	    // At setpoint
	    IF #Enabled = TRUE THEN
	        #sTag.bAtSetpoint := NOT(#sTag.bOutput);
	    ELSE
	        #sTag.bAtSetpoint := FALSE;
	    END_IF;
	
	    // Controller fault
	    #sTag.bFault := FALSE;
	
	END_IF;
	
	// Mode
	IF #sTag.bManualOverride = TRUE THEN
	    #sTag.nMode := 3;
	ELSIF #sTag.bEnable = TRUE THEN
	    #sTag.nMode := 1;
	ELSE
	    #sTag.nMode := 0;
	END_IF;
	
	// Local outputs
	#bOutput := #sTag.bOutput;
	#bAtSetpoint := #sTag.bAtSetpoint;
	
	
END_FUNCTION_BLOCK

FUNCTION_BLOCK "fbHysteresis2"   // FB64, LAD
TITLE = fbHysteresis2
{ S7_Optimized_Access := 'TRUE' }
AUTHOR : Heaten
VERSION : 0.1
// Hysteresis function with bool inputs
// stored: AutoNumber true, IsIECCheckEnabled false, IsRetainMemResEnabled false, MemoryReserve 0, SetENOAutomatically false, UDAEnableTagReadback false
   VAR_INPUT
      bEnable : Bool;
      bHigh : Bool;
      bLow : Bool;
      bAbove : Bool;
      bReset : Bool;
   END_VAR
   VAR_OUTPUT
      bOut : Bool;
   END_VAR
   VAR
      State : Bool;
   END_VAR
   VAR_TEMP
      bStartSignal : Bool;
      bStopSignal : Bool;
   END_VAR
BEGIN

REGION Network 1 (SCL): Polarity of the control
   // Above = 1: when process state is "high" eg cooling, emptying, depressurizing
   // Above = 0: when precess state is "low" eg heating, filling, pressurizing
   IF #bAbove = TRUE THEN
       // emptying, cooling, depressurizing etc
       #bStartSignal := #bHigh;
       #bStopSignal := NOT(#bLow);
   ELSE
       // filling, heating, pressurizing etc
       #bStartSignal := NOT(#bLow);
       #bStopSignal := #bHigh;
   END_IF;
END_REGION

REGION Network 2: Switch ouput
   // Initial state = OFF
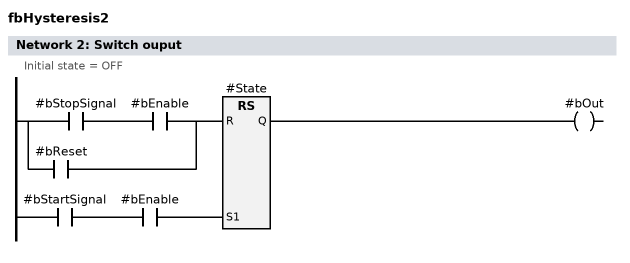
   RUNG wire#powerrail
      Contact( #bStopSignal )
      Contact( #bEnable )
      wire#w1
      S_RS(operand := #State, s1 := wire#w2)
      Coil( #bOut )
   END_RUNG
   RUNG wire#powerrail
      Contact( #bReset )
   END_RUNG wire#w1
   RUNG wire#powerrail
      Contact( #bStartSignal )
      Contact( #bEnable )
   END_RUNG wire#w2
   // the same network as SCL:
   IF (#bStopSignal AND #bEnable) OR #bReset THEN
       #State := FALSE;   // RS flip-flop
   END_IF;
   IF #bStartSignal AND #bEnable THEN #State := TRUE; END_IF;
   #bOut := #State;
END_REGION
END_FUNCTION_BLOCK

FUNCTION_BLOCK "ShaftSealCartridge"   // FB13, FBD
TITLE = Shaft seal cartridge
{ S7_Optimized_Access := 'TRUE' }
VERSION : 0.1
// stored: AutoNumber true, IsIECCheckEnabled false, IsRetainMemResEnabled false, MemoryReserve 100, SetENOAutomatically false, UDAEnableTagReadback false
   VAR_INPUT
      bEnable { ExternalAccessible := 'False'; ExternalVisible := 'False'; ExternalWritable := 'False'} : Bool;   // Enable from process. 1 = enabled, 0 = disabled.
      bReset { ExternalAccessible := 'False'; ExternalVisible := 'False'; ExternalWritable := 'False'} : Bool;
   END_VAR
   VAR
      Cooler { ExternalAccessible := 'False'; ExternalVisible := 'False'; ExternalWritable := 'False'} : "fbOnOffRegulator";
      Recharge { ExternalAccessible := 'False'; ExternalVisible := 'False'; ExternalWritable := 'False'; S7_SetPoint := 'True'} : "fbOnOffRegulator";
      A5257 { ExternalAccessible := 'False'; ExternalVisible := 'False'; ExternalWritable := 'False'; S7_SetPoint := 'True'} : "fbLowAlarm";
      A5258 { ExternalAccessible := 'False'; ExternalVisible := 'False'; ExternalWritable := 'False'; S7_SetPoint := 'True'} : "fbHighAlarm";
      A5259 { ExternalAccessible := 'False'; ExternalVisible := 'False'; ExternalWritable := 'False'; S7_SetPoint := 'True'} : "fbHighAlarm";
      A5260 { ExternalAccessible := 'False'; ExternalVisible := 'False'; ExternalWritable := 'False'; S7_SetPoint := 'True'} : "fbLowAlarm";
      A5261 { ExternalAccessible := 'False'; ExternalVisible := 'False'; ExternalWritable := 'False'; S7_SetPoint := 'True'} : "fbLowAlarm";
      A5262 { ExternalAccessible := 'False'; ExternalVisible := 'False'; ExternalWritable := 'False'; S7_SetPoint := 'True'} : "fbHighAlarm";
      A5263 { ExternalAccessible := 'False'; ExternalVisible := 'False'; ExternalWritable := 'False'; S7_SetPoint := 'True'} : "fbHighAlarm";
      A5268 { ExternalAccessible := 'False'; ExternalVisible := 'False'; ExternalWritable := 'False'; S7_SetPoint := 'True'} : "fbDigitalAlarm";
      nState { ExternalAccessible := 'False'; ExternalVisible := 'False'; ExternalWritable := 'False'; S7_SetPoint := 'True'} : USInt;
      bEnableAuto { ExternalAccessible := 'False'; ExternalVisible := 'False'; ExternalWritable := 'False'} : Bool;   // Circulation regulator is enabled in Auto
      bEnableCoolerAuto { ExternalAccessible := 'False'; ExternalVisible := 'False'; ExternalWritable := 'False'} : Bool;   // Cooling regulator is enabled in Auto
      bEnableRechargeAuto { ExternalAccessible := 'False'; ExternalVisible := 'False'; ExternalWritable := 'False'} : Bool;   // Recharging regulator is enabled in Auto
      bRunReqAuto { ExternalAccessible := 'False'; ExternalVisible := 'False'; ExternalWritable := 'False'} : Bool;   // Run in auto
      bStart { ExternalAccessible := 'False'; ExternalVisible := 'False'; ExternalWritable := 'False'} : R_TRIG;
   END_VAR
BEGIN

REGION Network 1: Delta-T over shaft seal
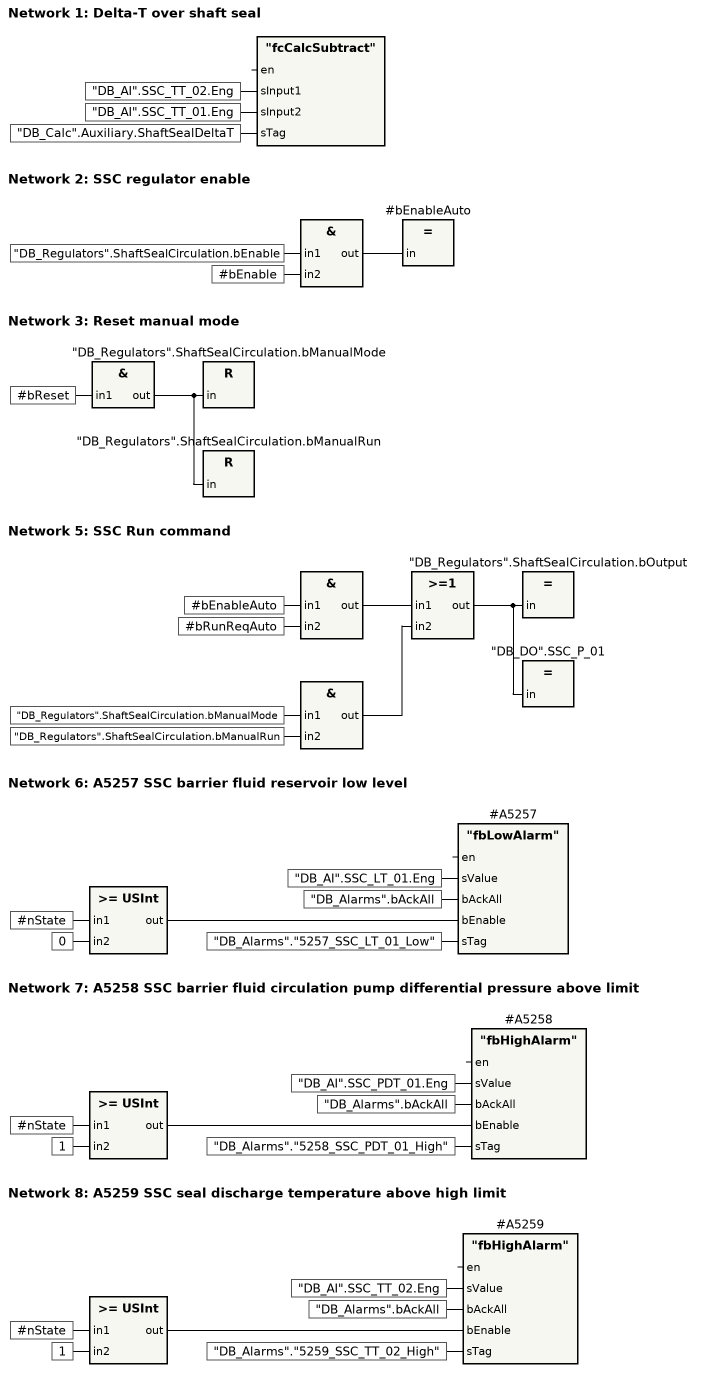
   "fcCalcSubtract"(sInput1 := "DB_AI".SSC_TT_02.Eng,
                    sInput2 := "DB_AI".SSC_TT_01.Eng,
                    sTag := "DB_Calc".Auxiliary.ShaftSealDeltaT);
END_REGION

REGION Network 2: SSC regulator enable
   // Start from input pin when enabled from HMI
   #bEnableAuto := "DB_Regulators".ShaftSealCirculation.bEnable AND #bEnable;
END_REGION

REGION Network 3: Reset manual mode
   IF #bReset THEN
       "DB_Regulators".ShaftSealCirculation.bManualMode := FALSE;
       "DB_Regulators".ShaftSealCirculation.bManualRun := FALSE;
   END_IF;
END_REGION

REGION Network 4 (SCL): SSC system state machine
   // Don't go into run state unless the pressure and temperature are first ok
   // Prevent retriggering
   #bStart(CLK := #bEnableAuto);

   CASE #nState OF

       0: // OFF
           #bEnableCoolerAuto := FALSE;
           #bEnableRechargeAuto := FALSE;
           #bRunReqAuto := FALSE;
           "DB_Regulators".ShaftSealCirculation.bFault := FALSE;
           IF #bStart.Q THEN
               #nState := 1;
           END_IF;
       1: // Startup. Wait for pressure and temperature to be ok
           #bEnableCoolerAuto := TRUE;
           #bEnableRechargeAuto := TRUE;
           //IF "DB_Regulators".ShaftSealCirculation.bEnable = FALSE THEN
           IF #bEnableAuto = FALSE THEN
               // Stop command
               #nState := 0;
           ELSIF "DB_Regulators".ShaftSealCirculation.bPressureLow AND "DB_Regulators".ShaftSealCirculation.bReservoirLow THEN
               // Barrier fluid pressure low and low fluid in recharge tank (can't recharge), give up.
               "DB_Regulators".ShaftSealCirculation.bFault := TRUE;
               #nState := 0;
           ELSIF "DB_Regulators".ShaftSealRecharge.bAtSetpoint AND "DB_Regulators".ShaftSealCooler.bAtSetpoint THEN
               // Pressure and temperature ok
               #nState := 2;
           END_IF;
       2: // Running
           #bRunReqAuto := TRUE;
           //IF "DB_Regulators".ShaftSealCirculation.bEnable = FALSE THEN
           IF #bEnableAuto = FALSE THEN
               // Stop command
               #nState := 0;
           END_IF;
           // Generate fault signal only in running state.
           "DB_Regulators".ShaftSealCirculation.bFault := "DB_Regulators".ShaftSealCirculation.bPressureLow OR "DB_Regulators".ShaftSealCirculation.bTemperatureHigh OR "DB_Regulators".ShaftSealCirculation.bDifferentialPressureHigh;
   END_CASE;
END_REGION

REGION Network 5: SSC Run command
   "DB_Regulators".ShaftSealCirculation.bOutput := (#bEnableAuto AND #bRunReqAuto) OR ("DB_Regulators".ShaftSealCirculation.bManualMode AND "DB_Regulators".ShaftSealCirculation.bManualRun);
   "DB_DO".SSC_P_01 := "DB_Regulators".ShaftSealCirculation.bOutput;
END_REGION

REGION Network 6: A5257 SSC barrier fluid reservoir low level
   // Always active
   #A5257(sValue := "DB_AI".SSC_LT_01.Eng,   // "fbLowAlarm"
          bAckAll := "DB_Alarms".bAckAll,
          bEnable := #nState >= 0,
          sTag := "DB_Alarms"."5257_SSC_LT_01_Low");
END_REGION

REGION Network 7: A5258 SSC barrier fluid circulation pump differential pressure above limit
   #A5258(sValue := "DB_AI".SSC_PDT_01.Eng,   // "fbHighAlarm"
          bAckAll := "DB_Alarms".bAckAll,
          bEnable := #nState >= 1,
          sTag := "DB_Alarms"."5258_SSC_PDT_01_High");
END_REGION

REGION Network 8: A5259 SSC seal discharge temperature above high limit
   #A5259(sValue := "DB_AI".SSC_TT_02.Eng,   // "fbHighAlarm"
          bAckAll := "DB_Alarms".bAckAll,
          bEnable := #nState >= 1,
          sTag := "DB_Alarms"."5259_SSC_TT_02_High");
END_REGION

REGION Network 9: A5260 SSC barrier fluid circulation pump suction temperature below low limit
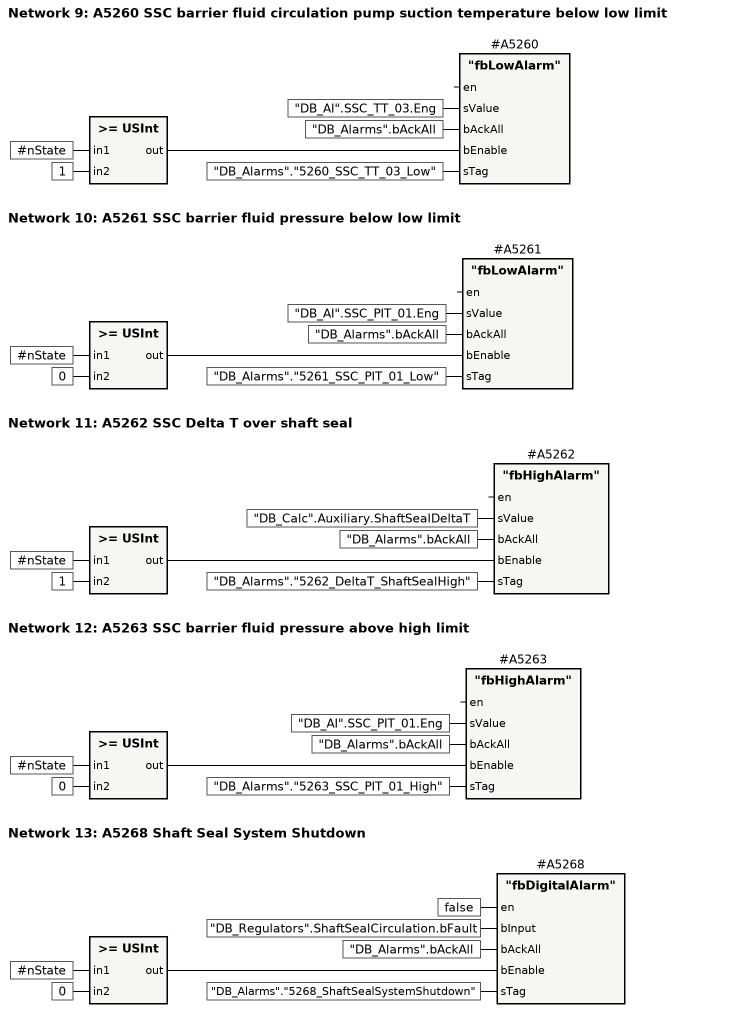
   #A5260(sValue := "DB_AI".SSC_TT_03.Eng,   // "fbLowAlarm"
          bAckAll := "DB_Alarms".bAckAll,
          bEnable := #nState >= 1,
          sTag := "DB_Alarms"."5260_SSC_TT_03_Low");
END_REGION

REGION Network 10: A5261 SSC barrier fluid pressure below low limit
   #A5261(sValue := "DB_AI".SSC_PIT_01.Eng,   // "fbLowAlarm"
          bAckAll := "DB_Alarms".bAckAll,
          bEnable := #nState >= 0,
          sTag := "DB_Alarms"."5261_SSC_PIT_01_Low");
END_REGION

REGION Network 11: A5262 SSC Delta T over shaft seal
   #A5262(sValue := "DB_Calc".Auxiliary.ShaftSealDeltaT,   // "fbHighAlarm"
          bAckAll := "DB_Alarms".bAckAll,
          bEnable := #nState >= 1,
          sTag := "DB_Alarms"."5262_DeltaT_ShaftSealHigh");
END_REGION

REGION Network 12: A5263 SSC barrier fluid pressure above high limit
   #A5263(sValue := "DB_AI".SSC_PIT_01.Eng,   // "fbHighAlarm"
          bAckAll := "DB_Alarms".bAckAll,
          bEnable := #nState >= 0,
          sTag := "DB_Alarms"."5263_SSC_PIT_01_High");
END_REGION

REGION Network 13: A5268 Shaft Seal System Shutdown
   // Regulator fault
   IF false THEN
       #A5268(bInput := "DB_Regulators".ShaftSealCirculation.bFault,   // "fbDigitalAlarm"
              bAckAll := "DB_Alarms".bAckAll,
              bEnable := #nState >= 0,
              sTag := "DB_Alarms"."5268_ShaftSealSystemShutdown");
   END_IF;
END_REGION

REGION Network 14: Faults
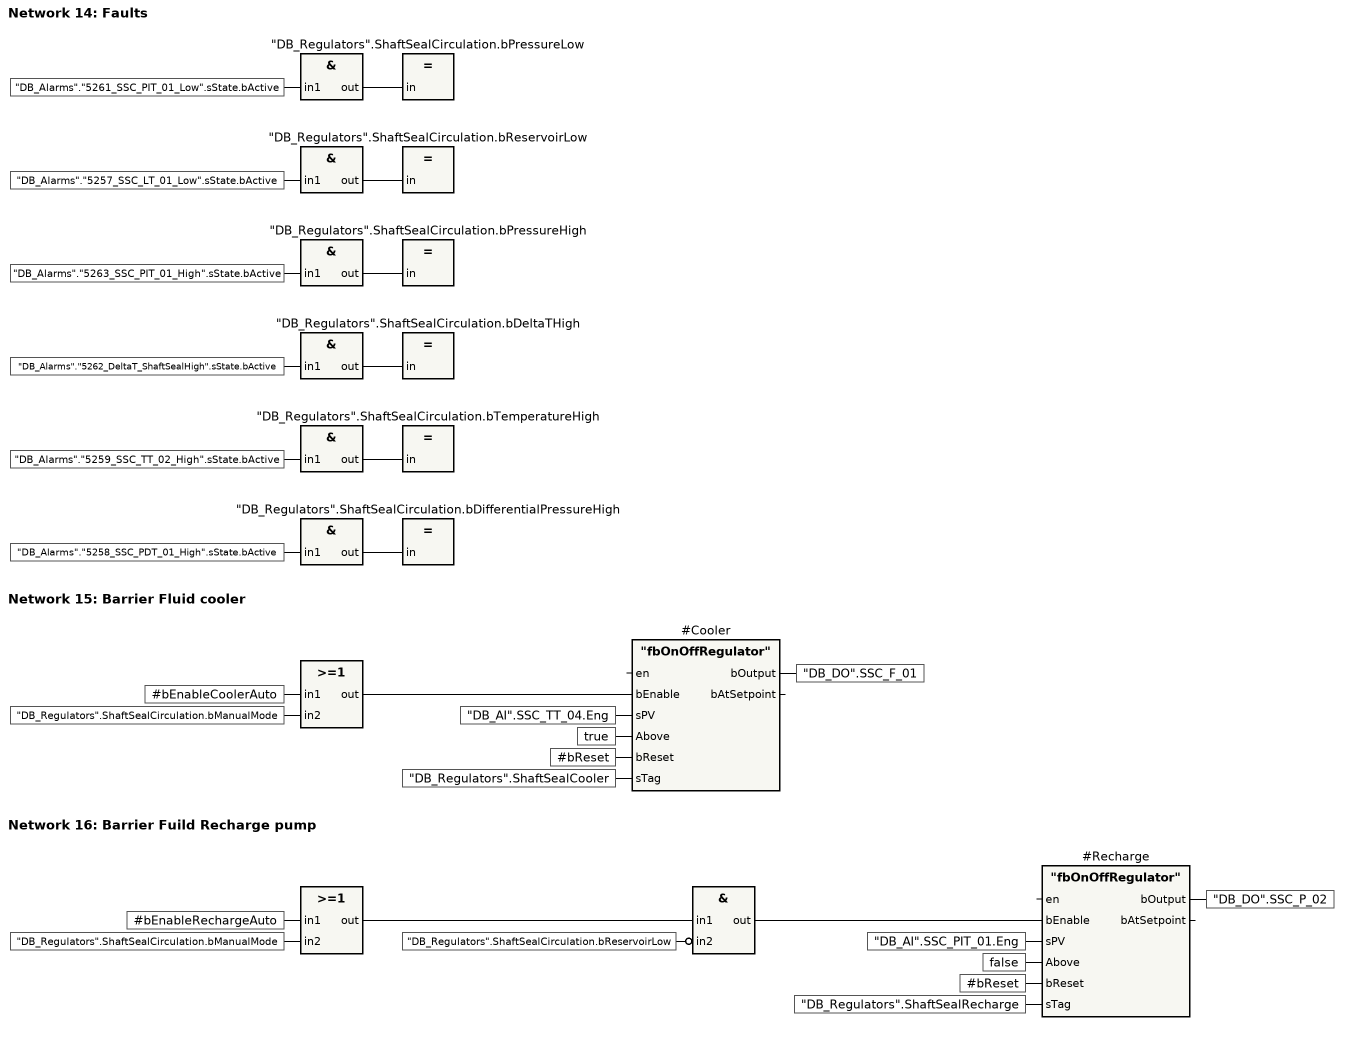
   "DB_Regulators".ShaftSealCirculation.bPressureLow := "DB_Alarms"."5261_SSC_PIT_01_Low".sState.bActive;
   "DB_Regulators".ShaftSealCirculation.bReservoirLow := "DB_Alarms"."5257_SSC_LT_01_Low".sState.bActive;
   "DB_Regulators".ShaftSealCirculation.bPressureHigh := "DB_Alarms"."5263_SSC_PIT_01_High".sState.bActive;
   "DB_Regulators".ShaftSealCirculation.bDeltaTHigh := "DB_Alarms"."5262_DeltaT_ShaftSealHigh".sState.bActive;
   "DB_Regulators".ShaftSealCirculation.bTemperatureHigh := "DB_Alarms"."5259_SSC_TT_02_High".sState.bActive;
   "DB_Regulators".ShaftSealCirculation.bDifferentialPressureHigh := "DB_Alarms"."5258_SSC_PDT_01_High".sState.bActive;
END_REGION

REGION Network 15: Barrier Fluid cooler
   // Run when the temperature in the barrier fluid gets too high
   #Cooler(bEnable := #bEnableCoolerAuto OR "DB_Regulators".ShaftSealCirculation.bManualMode,   // "fbOnOffRegulator"
           sPV := "DB_AI".SSC_TT_04.Eng,
           Above := true,
           bReset := #bReset,
           sTag := "DB_Regulators".ShaftSealCooler,
           bOutput => "DB_DO".SSC_F_01);
END_REGION

REGION Network 16: Barrier Fuild Recharge pump
   // Run when the pressure in the barrier fluid accumulator drops too low (and the reservoir is not empty)
   #Recharge(bEnable := (#bEnableRechargeAuto OR "DB_Regulators".ShaftSealCirculation.bManualMode) AND NOT "DB_Regulators".ShaftSealCirculation.bReservoirLow,   // "fbOnOffRegulator"
             sPV := "DB_AI".SSC_PIT_01.Eng,
             Above := false,
             bReset := #bReset,
             sTag := "DB_Regulators".ShaftSealRecharge,
             bOutput => "DB_DO".SSC_P_02);
END_REGION

REGION Network 17 (SCL)
   // Mode
   IF "DB_Regulators".ShaftSealCirculation.bManualMode = TRUE THEN
       "DB_Regulators".ShaftSealCirculation.nMode := 2;
   ELSIF "DB_Regulators".ShaftSealCirculation.bEnable = TRUE THEN
       "DB_Regulators".ShaftSealCirculation.nMode := 1;
   ELSE
       "DB_Regulators".ShaftSealCirculation.nMode := 0;
   END_IF;
END_REGION
END_FUNCTION_BLOCK

FUNCTION_BLOCK "LubricationPriming"   // FB20, FBD
{ S7_Optimized_Access := 'TRUE' }
VERSION : 0.1
// stored: AutoNumber true, IsIECCheckEnabled false, IsRetainMemResEnabled false, MemoryReserve 100, SetENOAutomatically false, UDAEnableTagReadback false
   VAR_INPUT
      bEnable { ExternalAccessible := 'False'; ExternalVisible := 'False'; ExternalWritable := 'False'} : Bool;
      bReset { ExternalAccessible := 'False'; ExternalVisible := 'False'; ExternalWritable := 'False'} : Bool;
   END_VAR
   VAR
      Pump { ExternalAccessible := 'False'; ExternalVisible := 'False'; ExternalWritable := 'False'} : "fbOnOffRegulator";
      Special { S7_SetPoint := 'True'} : "fbSpecialRegulator";
   END_VAR
   VAR_TEMP
      bOutput : Bool;
   END_VAR
BEGIN

REGION Network 1: Pump regulator
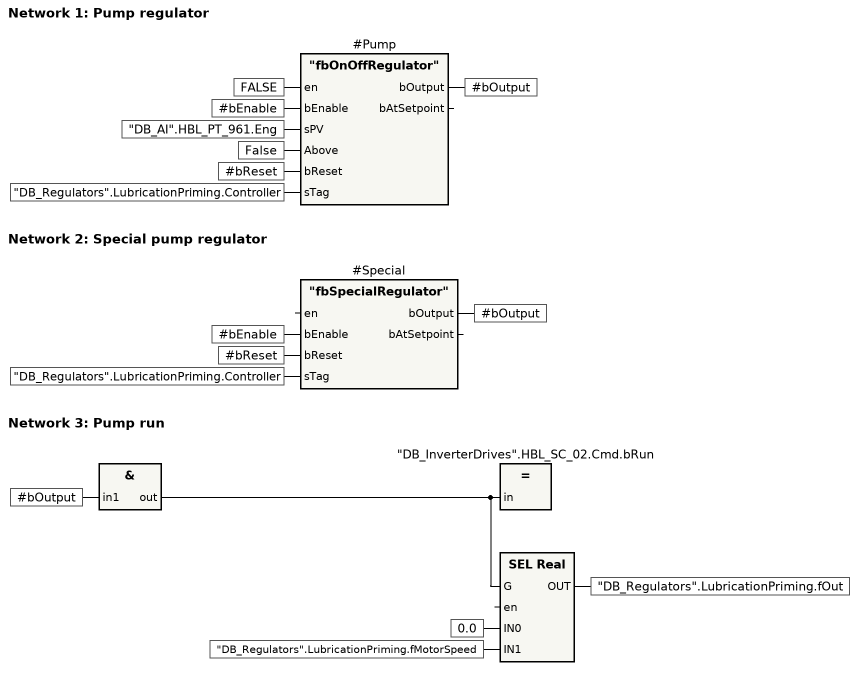
   IF FALSE THEN
       #Pump(bEnable := #bEnable,   // "fbOnOffRegulator"
             sPV := "DB_AI".HBL_PT_961.Eng,
             Above := False,
             bReset := #bReset,
             sTag := "DB_Regulators".LubricationPriming.Controller,
             bOutput => #bOutput);
   END_IF;
END_REGION

REGION Network 2: Special pump regulator
   // ##TEST: special situations require special regulators!
   #Special(bEnable := #bEnable,   // "fbSpecialRegulator"
            bReset := #bReset,
            sTag := "DB_Regulators".LubricationPriming.Controller,
            bOutput => #bOutput);
END_REGION

REGION Network 3: Pump run
   "DB_InverterDrives".HBL_SC_02.Cmd.bRun := #bOutput;
   "DB_Regulators".LubricationPriming.fOut := SEL(G := #bOutput, IN0 := 0.0, IN1 := "DB_Regulators".LubricationPriming.fMotorSpeed);
END_REGION

REGION Network 4: Inverter run
END_REGION
END_FUNCTION_BLOCK

FUNCTION_BLOCK "fbSpecialRegulator"
{ S7_Optimized_Access := 'TRUE' }
VERSION : 0.1
   VAR_INPUT 
      bEnable : Bool;   // Enable from process. 1 = enabled, 0 = disabled
      bReset : Bool;   // 1 = reset manual modes
   END_VAR

   VAR_OUTPUT 
      bOutput : Bool;
      bAtSetpoint : Bool;
   END_VAR

   VAR_IN_OUT 
      sTag : "stOnOffRegulator";
   END_VAR

   VAR 
      Dummy : Bool;
   END_VAR

   VAR_TEMP 
      fSetpoint : Real;
      Enabled : Bool;
   END_VAR


BEGIN
	// Special regulator.
	// Looks like an on/off regulator but in "Auto" mode, runs as soon as it is enabled. A kind of "null" regulator
	// The reason for still using this block is to allow all the other functions of the regulator, like the manual
	// override functions, and Reset, to still work. Not optimized, just a hack.
	// 
	
	// Reset manual modes.
	IF #bReset THEN
	    #sTag.bManualMode := FALSE;
	    #sTag.fManualSetpoint := 0.0;
	    #sTag.bManualOverride := FALSE;
	    #sTag.bOverrideCmd := FALSE;
	END_IF;
	
	IF #sTag.bManualOverride = TRUE THEN
	    // In manual override, everything is awesome
	    #sTag.bAtSetpoint := TRUE;
	    #sTag.bFault := FALSE;
	    #sTag.bOutput := #sTag.bOverrideCmd;
	ELSE
	    // Enabled when enabled from process and from HMI (Auto), no manual mode
	    #Enabled := (#bEnable AND #sTag.bEnable);
	
	    // Run controller
	    IF #Enabled = TRUE THEN
	        #sTag.bOutput := TRUE;
	    ELSE
	        #sTag.bOutput  := FALSE;
	    END_IF;
	    
	    #sTag.bAtSetpoint := NOT (#sTag.bOutput);
	    
	    // Controller fault
	    #sTag.bFault := FALSE;
	
	END_IF;
	
	// Mode
	IF #sTag.bManualOverride = TRUE THEN
	    #sTag.nMode := 3;
	ELSIF #sTag.bManualMode = TRUE THEN
	    #sTag.nMode := 2;
	ELSIF #sTag.bEnable = TRUE THEN
	    #sTag.nMode := 1;
	ELSE
	    #sTag.nMode := 0;
	END_IF;
	
	// Local outputs
	#bOutput := #sTag.bOutput;
	#bAtSetpoint := #sTag.bAtSetpoint;
	
	
END_FUNCTION_BLOCK

FUNCTION_BLOCK "fbPurgeControl"
{ S7_Optimized_Access := 'TRUE' }
AUTHOR : Heaten
VERSION : 0.1
   VAR_INPUT 
      bEnable : Bool;   // 1 = enable, 0 = disable
      bRotationStopped : Bool;   // 1 = rotation stopped, 0 = rotating
      DeltaP : "stCalcValue";   // [kPa] 
      Speed : "stCalcValue";   // [rpm]
      fCycleTime : Real;
   END_VAR

   VAR_OUTPUT 
      bPurging : Bool;
      bSpinning : Bool;
      bDone : Bool := false;
   END_VAR

   VAR_IN_OUT 
      sTag : "stPurgeControl";
   END_VAR

   VAR 
      nState : Int;   // 0 = Idle, 1 = Purge, 2 = Ramp up, 3 = Spin, 4 = Ramp down, 5 = Reset
      PurgeTimer {InstructionName := 'TON_TIME'; LibVersion := '1.0'; S7_SetPoint := 'False'} : TON_TIME;   // How long to purge for
      SpinTimer {InstructionName := 'TON_TIME'; LibVersion := '1.0'} : TON_TIME;   // How long to spin for
      PumpStartTimer {InstructionName := 'TON_TIME'; LibVersion := '1.0'} : TON_TIME;   // How long to wait for the pump to start & generate pressure
      tRamp : Time;   // Time to ramp up to spin speed
      tSpin : Time;   // Time at full spin speed
      Start {InstructionName := 'R_TRIG'; LibVersion := '1.0'; S7_SetPoint := 'False'} : R_TRIG;
   END_VAR

   VAR_TEMP 
      bEnabled : Bool;
   END_VAR

   VAR CONSTANT 
      PrimingDelay : Time := T#4s;
   END_VAR


BEGIN
	// Purge controller
	// Run a compressor purge cycle:
	// 1. Repeat x times: (where x can be zero)
	//    a. Drain the suction manifold. Either for a certain amount of time, or look at the deltaP over the pump
	//    b. Spin the compressor to get the suction line to barf up a slug of liquid, with configurable ramp, speed and duration
	// 2. Drain the suction manifold. Either for a certain amount of time, or look at the deltaP over the pump
	// 3. bDone = TRUE
	// NOTE: "look at the deltaP over the pump" means run the pump for #PrimingDelay, then continue as long as pump delta P is not less than 
	// sTag.Purge.fPurgeDeltaP
	
	// Enable. Edge trigger to run it only once. bReset is like a momentary disable
	#bEnabled := #bEnable AND #sTag.bEnable AND NOT #sTag.bReset;
	#Start(CLK := #bEnable AND #sTag.bEnable);
	
	// Be quiet when not in operation
	IF #bEnabled = FALSE THEN
	    #sTag.bDone := FALSE;
	END_IF;
	
	// Run timers outside of the state machine so they run & reset properly
	#PurgeTimer(IN := (#nState = 1 OR #nState = 6), PT := #sTag.Purge.tPurgeTime);
	#SpinTimer(IN := (#nState = 3), PT := #tSpin);
	#PumpStartTimer(IN := ((#nState = 1 OR #nState = 6) AND #sTag.Purge.nPurgeType = 1), PT := #PrimingDelay);
	
	// Purge sequencer
	CASE #nState OF
	    0: // Idle
	        IF #Start.Q = TRUE THEN
	            IF #sTag.nPurgeCycles = 0 THEN
	                #nState := 6;
	            ELSE
	                #sTag.nPurgeCyclesRemaining := #sTag.nPurgeCycles;
	                #sTag.bDone := FALSE;
	                #tRamp := UDINT_TO_TIME(REAL_TO_UDINT((#sTag.Spin.fSpinSpeed/#sTag.Spin.fSpinRamp)*1000));
	                #tSpin := #sTag.Spin.tSpinTime - 2 * #tRamp;
	                #nState := 1;
	            END_IF;
	        END_IF;
	    1: // Purge
	        IF #bEnabled = FALSE THEN
	            #nState := 5;
	        ELSE
	            // Start purging
	            #sTag.bPurging := TRUE;
	            // Decide when to stop
	            IF #sTag.Purge.nPurgeType = 0 THEN
	                // Timer
	                IF #PurgeTimer.Q = TRUE THEN
	                    #sTag.bPurging := FALSE;
	                    #nState := 2;
	                END_IF;
	            ELSIF #sTag.Purge.nPurgeType = 1 THEN
	                // Delta P
	                IF #PumpStartTimer.Q AND (#DeltaP.fValue < #sTag.Purge.fPurgeDeltaP) THEN
	                    #sTag.bPurging := FALSE;
	                    #nState := 2;
	                END_IF;
	            END_IF;
	        END_IF;
	    2: // Ramp Up
	        "RampLimiter"(InputValue            := #sTag.Spin.fSpinSpeed,                                  
	                      "PositivChange per_s" := #sTag.Spin.fSpinRamp,
	                      "NegativChange per_s" := -#sTag.Spin.fSpinRamp,
	                      fCycleTime            := #fCycleTime,
	                      OutputValue           := #sTag.fSpinOut);
	        IF #bEnabled = FALSE THEN
	            #nState := 5;
	        ELSIF #Speed.fValue > #sTag.Spin.fSpinSpeed - 5 THEN
	            #nState := 3;
	        END_IF;
	    3: // Spin
	        IF #bEnabled = FALSE THEN
	            #nState := 5;
	        ELSIF #SpinTimer.Q = TRUE THEN
	            #nState := 4;
	        END_IF;
	    4: // Ramp down
	        "RampLimiter"(InputValue            := 0.0,                         
	                      "PositivChange per_s" := #sTag.Spin.fSpinRamp,
	                      "NegativChange per_s" := -#sTag.Spin.fSpinRamp,
	                      fCycleTime            := #fCycleTime,
	                      OutputValue           := #sTag.fSpinOut);
	        IF #bEnabled = FALSE THEN
	            #nState := 5;
	        ELSIF #bRotationStopped = TRUE THEN
	            #sTag.fSpinOut := 0;
	            #sTag.nPurgeCyclesRemaining := #sTag.nPurgeCyclesRemaining - 1;
	            IF #sTag.nPurgeCyclesRemaining = 0 THEN
	                #nState := 6;
	            ELSE
	                #nState := 1;
	            END_IF;
	        END_IF;
	    5: // Reset
	        #sTag.nPurgeCyclesRemaining := 0;
	        #sTag.bPurging := FALSE;
	        #sTag.fSpinOut := 0;
	        #sTag.bDone := TRUE;
	        #nState := 0;
	    6: // Last purge
	        IF #bEnabled = FALSE THEN
	            #nState := 5;
	        ELSE
	            // Start purging
	            #sTag.bPurging := TRUE;
	            // Decide when to stop
	            IF #sTag.Purge.nPurgeType = 0 THEN
	                // Timer
	                IF #PurgeTimer.Q = TRUE THEN
	                    #sTag.bPurging := FALSE;
	                    #nState := 5;
	                END_IF;
	            ELSIF #sTag.Purge.nPurgeType = 1 THEN
	                // Delta P
	                IF #PumpStartTimer.Q AND (#DeltaP.fValue < #sTag.Purge.fPurgeDeltaP) THEN
	                    #sTag.bPurging := FALSE;
	                    #nState := 5;
	                END_IF;
	            END_IF;
	        END_IF;
	END_CASE;
	
	// Mode
	IF #sTag.bEnable = TRUE THEN
	    #sTag.nMode := 1;
	ELSE
	    #sTag.nMode := 0;
	END_IF;
	
	// Local outputs     
	#bDone := #sTag.bDone;
	#bPurging := #sTag.bPurging;
	#bSpinning := #sTag.bSpinning := (#nState = 2 OR #nState = 3 OR #nState = 4);
END_FUNCTION_BLOCK

FUNCTION_BLOCK "fbFilterDryer"   // FB53, FBD
TITLE = Periodic regulator with a fixed setpoint output
{ S7_Optimized_Access := 'TRUE' }
AUTHOR : Heaten
VERSION : 0.1
// stored: AutoNumber true, IsIECCheckEnabled false, IsRetainMemResEnabled false, MemoryReserve 0, SetENOAutomatically false, UDAEnableTagReadback false
   VAR_INPUT
      bEnable : Bool;
      bReset : Bool;
   END_VAR
   VAR_OUTPUT
      bOut : Bool;
      fOut : Real;
   END_VAR
   VAR_IN_OUT
      sTag : "stFilterDryer";
   END_VAR
   VAR
      Controller : "fbPeriodicRegulator";
   END_VAR
   VAR_TEMP
      bOutput_1 : Bool;
   END_VAR
BEGIN

REGION Network 1: Run regulator
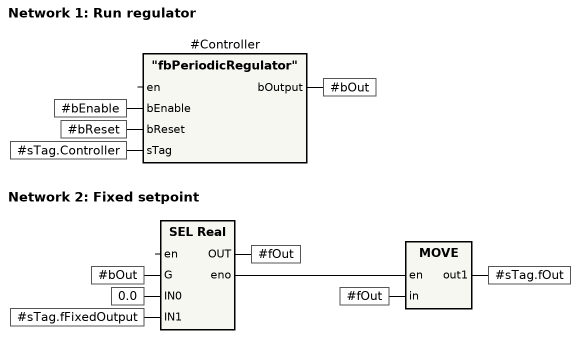
   #Controller(bEnable := #bEnable, bReset := #bReset, sTag := #sTag.Controller, bOutput => #bOut);   // "fbPeriodicRegulator"
END_REGION

REGION Network 2: Fixed setpoint
   // ENO of a box is taken as its EN; it also drops when the box reports an error
   #fOut := SEL(G := #bOut, IN0 := 0.0, IN1 := #sTag.fFixedOutput);
   #sTag.fOut := #fOut;
END_REGION
END_FUNCTION_BLOCK

FUNCTION_BLOCK "fbPeriodicRegulator"
{ S7_Optimized_Access := 'TRUE' }
AUTHOR : Heaten
VERSION : 0.1
   VAR_INPUT 
      bEnable : Bool;   // 1 = enable regulator, 0 = disable regulator
      bReset : Bool;   // 1 = reset everything to zero
   END_VAR

   VAR_OUTPUT 
      bOutput : Bool;
   END_VAR

   VAR_IN_OUT 
      sTag : "stPeriodicRegulator";
   END_VAR

   VAR 
      Controller { S7_SetPoint := 'False'} : "fbPWMController";
   END_VAR

   VAR_TEMP 
      Enabled : Bool;
   END_VAR


BEGIN
	// Periodic regulator
	// Periodic control of an output. Also called timer-based control.
	// The on-period and total period are parameters
	// Auto mode: periodic operation when Enable = true
	// Manual override: force the output on or off
	// 
	
	// Reset manual modes.
	IF #bReset THEN
	    #sTag.bManualOverride := FALSE;
	    #sTag.bOverrideCmd := FALSE;
	    #Controller.bEnable := FALSE;
	END_IF;
	
	// Select operating mode
	IF #sTag.bManualOverride = TRUE THEN
	    // In manual override, everything is awesome
	    #sTag.bFault := FALSE;
	    #sTag.bOutput := #sTag.bOverrideCmd;
	ELSE
	    // Enabled when enabled from process and from HMI (Auto)
	    #Enabled := (#bEnable AND #sTag.bEnable);
	    
	    // Run controller
	    #Controller(bEnable := #Enabled,
	                tOnTime := #sTag.tOnTime,
	                tPeriod := #sTag.tPeriod,
	                bOut => #sTag.bOutput,
	                tOnTimeElapsed => #sTag.tOnTimeElapsed,
	                tPeriodElapsed => #sTag.tPeriodElapsed);
	    
	    // Controller fault
	    #sTag.bFault := FALSE;
	    
	END_IF;
	
	// Mode
	IF #sTag.bManualOverride = TRUE THEN
	    #sTag.nMode := 3;
	ELSIF #sTag.bEnable = TRUE THEN
	    #sTag.nMode := 1;
	ELSE
	    #sTag.nMode := 0;
	END_IF;
	
	// Local outputs
	#bOutput := #sTag.bOutput;
END_FUNCTION_BLOCK

FUNCTION_BLOCK "fbOilRecovery"   // FB58, FBD
TITLE = Run once every X times with a fixed valve setpoint
{ S7_Optimized_Access := 'TRUE' }
AUTHOR : Heaten
VERSION : 0.1
// stored: AutoNumber true, IsIECCheckEnabled false, IsRetainMemResEnabled false, MemoryReserve 0, SetENOAutomatically false, UDAEnableTagReadback false
   VAR_INPUT
      bEnable : Bool;
      bReset : Bool;
   END_VAR
   VAR_OUTPUT
      bOut : Bool;
      fOut : Real;
   END_VAR
   VAR_IN_OUT
      sTag : "stOilRecovery";
   END_VAR
   VAR
      Controller : "fbOneShotRegulator";
      epEnabled : R_TRIG;
      RunCounter { S7_SetPoint := 'True'} : UInt;
      RunCounterMod : UInt;
   END_VAR
   VAR RETAIN
      Count { S7_SetPoint := 'True'} : Bool;
   END_VAR
   VAR_TEMP
      bEnabled : Bool;
   END_VAR
BEGIN

REGION Network 1: Run signal
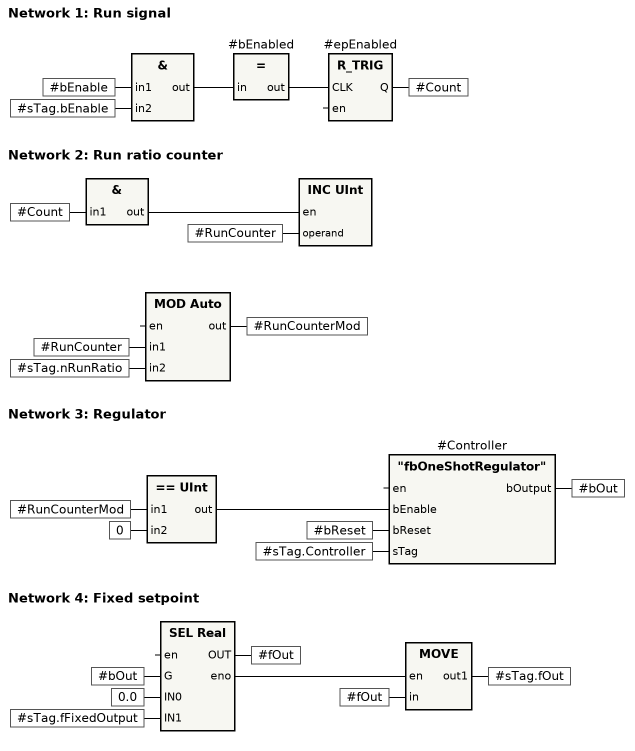
   #bEnabled := #bEnable AND #sTag.bEnable;
   #epEnabled(CLK := #bEnabled, Q => #Count);   // R_TRIG
END_REGION

REGION Network 2: Run ratio counter
   IF #Count THEN #RunCounter := #RunCounter + 1; END_IF;
   #RunCounterMod := #RunCounter MOD #sTag.nRunRatio;
END_REGION

REGION Network 3: Regulator
   // RunCounterMod is 0 every nth count.
   #Controller(bEnable := #RunCounterMod = 0, bReset := #bReset, sTag := #sTag.Controller, bOutput => #bOut);   // "fbOneShotRegulator"
END_REGION

REGION Network 4: Fixed setpoint
   // ENO of a box is taken as its EN; it also drops when the box reports an error
   #fOut := SEL(G := #bOut, IN0 := 0.0, IN1 := #sTag.fFixedOutput);
   #sTag.fOut := #fOut;
END_REGION
END_FUNCTION_BLOCK

FUNCTION_BLOCK "fbOneShotRegulator"
{ S7_Optimized_Access := 'TRUE' }
AUTHOR : Heaten
VERSION : 0.1
   VAR_INPUT 
      bEnable : Bool;   // 1 = enable regulator, 0 = disable regulator
      bReset : Bool;   // 1 = reset everything to zero
   END_VAR

   VAR_OUTPUT 
      bOutput : Bool;
   END_VAR

   VAR_IN_OUT 
      sTag : "stOneShotRegulator";
   END_VAR

   VAR 
      Controller { S7_SetPoint := 'False'} : "fbOneShot";
   END_VAR

   VAR_TEMP 
      Enabled : Bool;
   END_VAR


BEGIN
	// One-shot regulator
	// Activate something once for a certain period, with a start delay
	// The on-period and start delay are parameters
	// Auto mode: one-shot operation when Enable = true
	// Manual override: force the output on or off
	// 
	
	// Reset manual modes.
	IF #bReset THEN
	    #sTag.bManualOverride := FALSE;
	    #sTag.bOverrideCmd := FALSE;
	    #Controller.bEnable := FALSE;
	END_IF;
	
	// Select operating mode
	IF #sTag.bManualOverride = TRUE THEN
	    // In manual override, everything is awesome
	    #sTag.bFault := FALSE;
	    #sTag.bOutput := #sTag.bOverrideCmd;
	ELSE
	    // Enabled when enabled from process and from HMI (Auto)
	    #Enabled := (#bEnable AND #sTag.bEnable);
	    
	    // Run controller
	    #Controller(bEnable := #Enabled,
	                tOnTime := #sTag.tOnTime,
	                tStartDelay := #sTag.tStartDelay,
	                bOut => #sTag.bOutput,
	                tOnTimeElapsed => #sTag.tOnTimeElapsed,
	                tStartDelayElapsed => #sTag.tStartDelayElapsed);
	    
	    // Controller fault
	    #sTag.bFault := FALSE;
	    
	END_IF;
	
	// Mode
	IF #sTag.bManualOverride = TRUE THEN
	    #sTag.nMode := 3;
	ELSIF #sTag.bEnable = TRUE THEN
	    #sTag.nMode := 1;
	ELSE
	    #sTag.nMode := 0;
	END_IF;
	
	// Local outputs
	#bOutput := #sTag.bOutput;
END_FUNCTION_BLOCK

FUNCTION_BLOCK "fbOneShot"   // FB56, FBD
TITLE = One-shot with trigger delay
{ S7_Optimized_Access := 'TRUE' }
AUTHOR : Heaten
VERSION : 0.1
// stored: AutoNumber true, IsIECCheckEnabled false, IsRetainMemResEnabled false, MemoryReserve 0, SetENOAutomatically false, UDAEnableTagReadback false
   VAR_INPUT
      bEnable : Bool;   // 1 = enable controller, 0 = disable
      tOnTime : Time;
      tStartDelay : Time;
   END_VAR
   VAR_OUTPUT
      bOut : Bool;
      tOnTimeElapsed : Time;
      tStartDelayElapsed : Time;
   END_VAR
   VAR
      StartDelayTimer : TON_TIME;
      OnTimer { S7_SetPoint := 'True'} : TP_TIME;
   END_VAR
BEGIN

REGION Network 1: Trigger delay
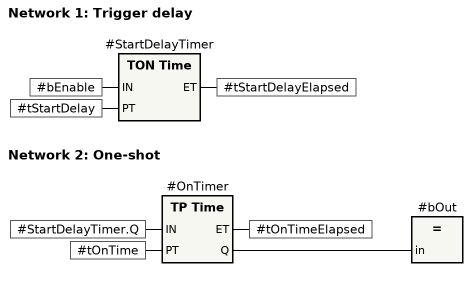
   #StartDelayTimer(IN := #bEnable, PT := #tStartDelay, ET => #tStartDelayElapsed);   // TON
END_REGION

REGION Network 2: One-shot
   #OnTimer(IN := #StartDelayTimer.Q, PT := #tOnTime, ET => #tOnTimeElapsed);   // TP
   #bOut := #OnTimer.Q;
END_REGION
END_FUNCTION_BLOCK

FUNCTION_BLOCK "fbNullRegulator"   // FB59, FBD
TITLE = PI Regulator
{ S7_Optimized_Access := 'TRUE' }
VERSION : 0.1
// stored: AutoNumber true, IsIECCheckEnabled false, IsRetainMemResEnabled false, MemoryReserve 0, SetENOAutomatically false, UDAEnableTagReadback false
   VAR_INPUT
      bEnable : Bool;
      bReset : Bool;
   END_VAR
   VAR_OUTPUT
      fOut : Real;
      bAtMin : Bool;
      bAtMax : Bool;
   END_VAR
   VAR_IN_OUT
      sTag : "stNullRegulator";
   END_VAR
   VAR
      Dummy : Real;
   END_VAR
   VAR_TEMP
      Enabled : Bool;
      fSelectedSetpoint : Real;
   END_VAR
BEGIN

REGION Network 1: Reset manual mode
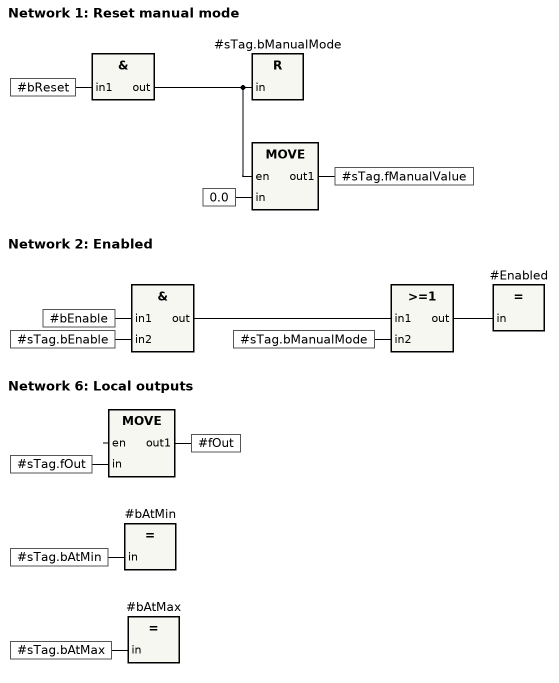
   IF #bReset THEN
       #sTag.bManualMode := FALSE;
       #sTag.fManualValue := 0.0;
   END_IF;
END_REGION

REGION Network 2: Enabled
   // Local input is from process control logic: when to run the regulator
   // Tag input is from HMI: do we want to run this regulator at all
   #Enabled := (#bEnable AND #sTag.bEnable) OR #sTag.bManualMode;
END_REGION

REGION Network 3 (SCL): Output selection
   IF #sTag.bManualMode = TRUE THEN
       #fSelectedSetpoint := #sTag.fManualValue;
   ELSE
       #fSelectedSetpoint := #sTag.fSetpoint;
   END_IF;

   #sTag.fOut := LIMIT(MN := #sTag.fOutMin, IN := #fSelectedSetpoint, MX := #sTag.fOutMax);
   #sTag.bAtMin := #sTag.fOut = #sTag.fOutMin;
   #sTag.bAtMax := #sTag.fOut = #sTag.fOutMax;
END_REGION

REGION Network 4 (SCL): Disable
   // This could be combined with logic above, and one day it might be!
   IF #Enabled = FALSE OR #sTag.bFault = TRUE THEN
       #sTag.fOut := 0.0;
       #sTag.bAtMin := FALSE;
       #sTag.bAtMax := FALSE;
   END_IF;
END_REGION

REGION Network 5 (SCL): Mode
   // Mode
   IF #sTag.bManualMode = TRUE THEN
       #sTag.nMode := 2;
   ELSIF #sTag.bEnable = TRUE THEN
       #sTag.nMode := 1;
   ELSE
       #sTag.nMode := 0;
   END_IF;
END_REGION

REGION Network 6: Local outputs
   #fOut := #sTag.fOut;
   #bAtMin := #sTag.bAtMin;
   #bAtMax := #sTag.bAtMax;
END_REGION
END_FUNCTION_BLOCK

FUNCTION_BLOCK "fbTrackingRegulator"
{ S7_Optimized_Access := 'TRUE' }
AUTHOR : Heaten
VERSION : 0.1
   VAR_INPUT 
      bEnable : Bool;
      bReset : Bool;
      sSP : "stCalcValue";   // Setpoint
      sPV : "stCalcValue";   // Process value
      sVelocity : "stCalcValue";   // Process value velocity
      fCycleTime : Real;
   END_VAR

   VAR_OUTPUT 
      fOut : Real;
      bAtMin : Bool;
      bAtMax : Bool;
   END_VAR

   VAR_IN_OUT 
      sTag : "stTrackingRegulator";
   END_VAR

   VAR 
      fStepsizePositive : Real;   // Output increment
      fStepsizeNegative : Real;   // Output decrement
   END_VAR

   VAR_TEMP 
      Enabled : Bool;
   END_VAR


BEGIN
	// Tracking regulator, a varaint of incremental control
	// Based on the "tracking ADC" algorithm, also known as "delta-encoded" or "counter-ramp"
	// The main parameters are the positive and negative slew rates. These control how big the increment in the output is.
	// The output is a staircase waveform which ramps the actuator up and down. The step size is calculated from the slew rate and cycle time.
	// There are two rates: the rate of change of the process value, and the rate of change of the actuator
	// For example, limiting the slew rate of a valve to keep the temperature increase below a limit
	
	// Detailed algorithm:
	// IF temperature < target AND temperature rate of change < positive limit THEN
	//    Increase valve output by positive step size
	// ELSIF temperature > target OR temperature rate of change > positive limit THEN
	//    Decrease valve output by negative step size
	// ELSE
	//    Keep valve output the same
	// END_IF
	// 
	
	// Tuning procedure:
	// 1. Set the fSlewRatePositive to something conservative like 0.2C/s
	// 2. Start HB and let it get to State 2
	// 3. Watch the heating of the steam condensers
	// 4. If the heating is very slow....
	
	// Copy to tag
	#sTag.fPV := #sPV.fValue;
	#sTag.fSP := #sSP.fValue;
	#sTag.fPVvelocity := #sVelocity.fValue;
	
	IF #bReset = TRUE THEN
	    #sTag.fOut := 0.0;
	    #sTag.bManualMode := FALSE;
	    #sTag.fManualValue := 0.0;
	END_IF;
	
	#Enabled := (#bEnable AND #sTag.bEnable) OR #sTag.bManualMode;
	
	// Step sizes
	#fStepsizePositive := #sTag.fSlewRatePositive / #fCycleTime;
	#fStepsizeNegative := #sTag.fSlewRateNegative / #fCycleTime;
	
	// Controller fault
	#sTag.bFault := #sSP.bError OR #sPV.bError OR #sVelocity.bError;
	
	IF #sTag.bManualMode = TRUE THEN
	    // Manual mode
	    #sTag.fOut := #sTag.fManualValue;
	ELSE
	    // Auto mode
	    IF #sPV.fValue < (#sSP.fValue - #sTag.fHysteresis) AND #sVelocity.fValue < #sTag.fVelocityPositiveLimit THEN
	        // Increase valve output
	        #sTag.fOut := #sTag.fOut + #fStepsizePositive;
	        #sTag.bAtSetpoint := FALSE;
	    ELSIF #sPV.fValue > (#sSP.fValue + #sTag.fHysteresis) OR #sVelocity.fValue > #sTag.fVelocityPositiveLimit THEN
	        // Decrease valve output
	        #sTag.fOut := #sTag.fOut - #fStepsizeNegative;
	        #sTag.bAtSetpoint := FALSE;
	    ELSE
	        // Keep valve output the same. Dummy branch but important to see the flow
	        #sTag.fOut := #sTag.fOut;
	        #sTag.bAtSetpoint := TRUE;
	    END_IF;
	END_IF;
	
	// Post processing
	IF #Enabled = FALSE OR #sTag.bFault = TRUE THEN
	    #sTag.fOut := 0.0;
	    #sTag.bAtMin := FALSE;
	    #sTag.bAtMax := FALSE;
	ELSE
	    //Evaluate limits exceeded first...
	    #sTag.bAtMin := NOT (#sTag.fOut > #sTag.fOutMin);
	    #sTag.bAtMax := #sTag.fOut >= #sTag.fOutMax;
	    //...before doing the actual limiting
	    #sTag.fOut := LIMIT(MN := #sTag.fOutMin, IN := #sTag.fOut, MX := #sTag.fOutMax);
	END_IF;
	
	// Mode
	IF #sTag.bManualMode = TRUE THEN
	    #sTag.nMode := 2;
	ELSIF #sTag.bEnable = TRUE THEN
	    #sTag.nMode := 1;
	ELSE
	    #sTag.nMode := 0;
	END_IF;
	
	// Local outputs
	#fOut := #sTag.fOut;
	#bAtMin := #sTag.bAtMin;
	#bAtMax := #sTag.bAtMax;
	
	
END_FUNCTION_BLOCK

FUNCTION_BLOCK "fbPIP_Regulator"   // FB28, FBD
TITLE = Position-velocity regulator (PI-P form)
{ S7_Optimized_Access := 'TRUE' }
AUTHOR : Heaten
VERSION : 0.1
// stored: AutoNumber true, IsIECCheckEnabled false, IsRetainMemResEnabled false, MemoryReserve 0, SetENOAutomatically false, UDAEnableTagReadback false
   VAR_INPUT
      sPV : "stCalcValue";   // Process value (position)
      sPVvel : "stCalcValue";   // Process value (velocity)
      fFeedback : Real;   // Output feedback (eg valve %, motor rpm)
      fCycleTime : Real;
      bEnable : Bool;
      bReset : Bool;
   END_VAR
   VAR_OUTPUT
      fOut : Real;
      bAtMin : Bool;
      bAtMax : Bool;
   END_VAR
   VAR_IN_OUT
      sTag : "stPIP_Regulator";
   END_VAR
   VAR
      Outer : Struct   // Outer loop = PI control
         D_Mem : Real;
         I_Mem : Real;
         Param_Mem : Real;
      END_STRUCT;
      Inner : Struct   // Inner loop = P control
         D_Mem : Real;
         I_Mem : Real;
         Param_Mem : Real;
      END_STRUCT;
      fSPVel : Real;
   END_VAR
   VAR_TEMP
      Enabled : Bool;
      fDeviation : Real;
      fDeviationVel : Real;
      bPI_AtMax : Bool;
      bPI_AtMin : Bool;
   END_VAR
BEGIN

REGION Network 1 (SCL): Comments and history
   // Position-velocity controller, cascaded PI-P form
   // 
   //                ___   pos   ____   vel   ___   vel   ___   out   __________         ______
   // pos ref ----> | Σ | ----> | PI | ----> | Σ | ----> | P | ----> | Actuator | ----> | Load |
   //             + |___| error |____|  ref  |___| error |___|       |__________|       |______|
   //                 ^ -                      ^ -                    _______               | 
   //                 |                        |_____________________| dP/dt |______________| measured velocity
   //                 |                                              |_______|              |
   //                 |_____________________________________________________________________| measured position
   //                 
   // For example, heating up a heat exchanger to a certain temperature without exceeding the temperature rise limit
   // 
   // Tuning Steps
   //
   // 1. Set the P constants of both controllers equal to 0, and integral to 9999. By default, the integral limit of the velocity
   //    controller should be set to the actuator's maximum position (eg 100%), and the integral limit of position
   //    controller should be set to the process max velocity (eg 5K/min).
   //
   // Important:from this step forth, the step response of position controller should always be evaluated.
   //
   // 2. Tune the KpVel parameter of the velocity controller. Increase the Kp of both position and velocity 
   //    controllers with a ratio of 10 (Kp_velocity = 10 * Kp_position). Once the real position starts to follow the
   //    reference position, stop increasing the Kp_position and only focus on increasing the Kp_velocity. Increase
   //    (sharpen) the velocity controller as much as possible. As a rule of thumb, increase kP_velocity until you get
   //    close to the instability margin (at this margin, you will feel a vibration effect and some acoustic noise
   //    which is because of controller sharpness). Now, you can reduce kP_velocity to 90% of its value to increase 
   //    the stability margin, and remove vibration noise.
   // 
   // 3. Now that the velocity controller is tuned, it is time to tune the parameters of the PID position 
   //    controller. Start with kP_position, and increase it until you again get close to the instability margin, and 
   //    then reduce kP_position to its 90%. So far, the proportional parts of both inner velocity loop and outer 
   //    position loop are tuned.
   //
   // 4. In this step, increase kI to eliminate the steady state error. As a suggestion start with kI equal to
   //    0.01, and in each step, increase it with a factor of 2. Increase kI step by step until the following two 
   //    conditions are met at the same time: - the overshoot is in its acceptable range - the steady-state error is 
   //    eliminated in a short enough period of time.
END_REGION

REGION Network 3: Reset manual mode
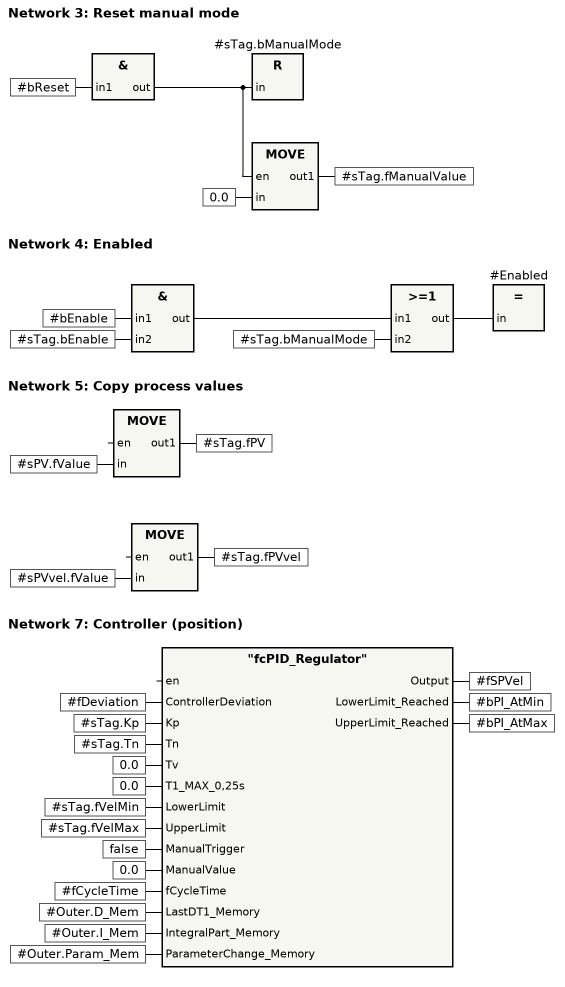
   IF #bReset THEN
       #sTag.bManualMode := FALSE;
       #sTag.fManualValue := 0.0;
   END_IF;
END_REGION

REGION Network 4: Enabled
   // Local input is from process control logic: when to run the regulator
   // Tag input is from HMI: do we want to run this regulator at all
   #Enabled := (#bEnable AND #sTag.bEnable) OR #sTag.bManualMode;
END_REGION

REGION Network 5: Copy process values
   #sTag.fPV := #sPV.fValue;
   #sTag.fPVvel := #sPVvel.fValue;
END_REGION

REGION Network 6 (SCL): Deviation (position)
   // NaN detection
   IF "isNaN"(#sTag.fSP) OR "isNaN"(#sTag.fPV) THEN
       #fDeviation := 0.0;
       #sTag.bFault := TRUE;
   ELSE
       #fDeviation := #sTag.fSP - #sTag.fPV;
       #sTag.bFault := FALSE;
   END_IF;
END_REGION

REGION Network 7: Controller (position)
   // NOTE: controller always runs regardless of mode.
   // This stage generates a velocity setpoint from the position error.
   // Max & min limits are of VELOCITY, this is not abug.
   "fcPID_Regulator"(ControllerDeviation := #fDeviation,
                     Kp := #sTag.Kp,
                     Tn := #sTag.Tn,
                     Tv := 0.0,
                     "T1_MAX_0,25s" := 0.0,
                     LowerLimit := #sTag.fVelMin,
                     UpperLimit := #sTag.fVelMax,
                     ManualTrigger := false,
                     ManualValue := 0.0,
                     fCycleTime := #fCycleTime,
                     LastDT1_Memory := #Outer.D_Mem,
                     IntegralPart_Memory := #Outer.I_Mem,
                     ParameterChange_Memory := #Outer.Param_Mem,
                     Output => #fSPVel,
                     LowerLimit_Reached => #bPI_AtMin,
                     UpperLimit_Reached => #bPI_AtMax);
END_REGION

REGION Network 8 (SCL): Deviation (velocity)
   // NaN detection
   IF "isNaN"(#sTag.fPVvel) THEN
       #fDeviationVel := 0.0;
       #sTag.bFault := TRUE;
   ELSE
       #fDeviationVel := #fSPVel - #sTag.fPVvel;
       #sTag.bFault := FALSE;
   END_IF;
END_REGION

REGION Network 9: Controller (velocity)
   // NOTE: controller always runs regardless of mode
   // This stage generates the manipulated value from the velocity error.
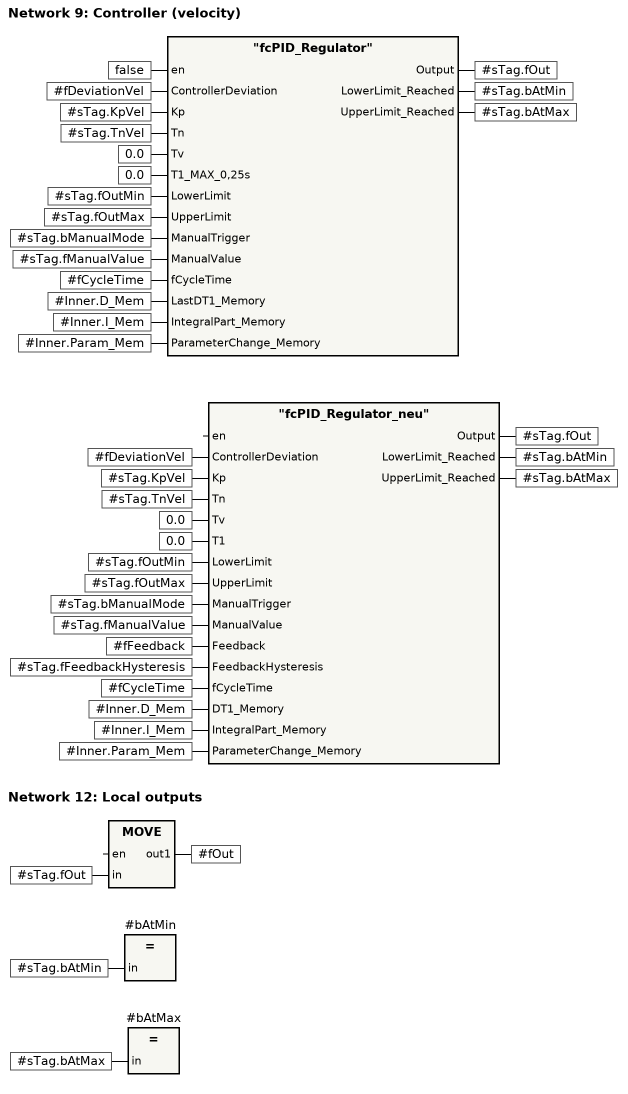
   IF false THEN
       "fcPID_Regulator"(ControllerDeviation := #fDeviationVel,
                         Kp := #sTag.KpVel,
                         Tn := #sTag.TnVel,
                         Tv := 0.0,
                         "T1_MAX_0,25s" := 0.0,
                         LowerLimit := #sTag.fOutMin,
                         UpperLimit := #sTag.fOutMax,
                         ManualTrigger := #sTag.bManualMode,
                         ManualValue := #sTag.fManualValue,
                         fCycleTime := #fCycleTime,
                         LastDT1_Memory := #Inner.D_Mem,
                         IntegralPart_Memory := #Inner.I_Mem,
                         ParameterChange_Memory := #Inner.Param_Mem,
                         Output => #sTag.fOut,
                         LowerLimit_Reached => #sTag.bAtMin,
                         UpperLimit_Reached => #sTag.bAtMax);
   END_IF;
   "fcPID_Regulator_neu"(ControllerDeviation := #fDeviationVel,
                         Kp := #sTag.KpVel,
                         Tn := #sTag.TnVel,
                         Tv := 0.0,
                         T1 := 0.0,
                         LowerLimit := #sTag.fOutMin,
                         UpperLimit := #sTag.fOutMax,
                         ManualTrigger := #sTag.bManualMode,
                         ManualValue := #sTag.fManualValue,
                         Feedback := #fFeedback,
                         FeedbackHysteresis := #sTag.fFeedbackHysteresis,
                         fCycleTime := #fCycleTime,
                         DT1_Memory := #Inner.D_Mem,
                         IntegralPart_Memory := #Inner.I_Mem,
                         ParameterChange_Memory := #Inner.Param_Mem,
                         Output => #sTag.fOut,
                         LowerLimit_Reached => #sTag.bAtMin,
                         UpperLimit_Reached => #sTag.bAtMax);
END_REGION

REGION Network 10 (SCL): Disable
   IF #Enabled = FALSE OR #sTag.bFault = TRUE THEN
       #sTag.fOut := 0.0;
       #sTag.bAtMin := FALSE;
       #sTag.bAtMax := FALSE;
   END_IF;
END_REGION

REGION Network 11 (SCL): Mode
   // Mode
   IF #sTag.bManualMode = TRUE THEN
       #sTag.nMode := 2;
   ELSIF #sTag.bEnable = TRUE THEN
       #sTag.nMode := 1;
   ELSE
       #sTag.nMode := 0;
   END_IF;
END_REGION

REGION Network 12: Local outputs
   #fOut := #sTag.fOut;
   #bAtMin := #sTag.bAtMin;
   #bAtMax := #sTag.bAtMax;
END_REGION
END_FUNCTION_BLOCK

FUNCTION_BLOCK "MotorControl"
{ S7_Optimized_Access := 'TRUE' }
VERSION : 0.1
   VAR_INPUT 
      PerformanceSetpoint { ExternalAccessible := 'False'; ExternalVisible := 'False'; ExternalWritable := 'False'} : Real;   // [%] Performance rate
      FastStop { ExternalAccessible := 'False'; ExternalVisible := 'False'; ExternalWritable := 'False'} : Bool;   // 1 = execute a fast stop, 0 = do nothing
   END_VAR

   VAR 
      NEngineRequest { ExternalAccessible := 'False'; ExternalVisible := 'False'; ExternalWritable := 'False'} : Real;   // [rpm]
      NEngineSetpoint { ExternalAccessible := 'False'; ExternalVisible := 'False'; ExternalWritable := 'False'} : Real;   // [rpm]
      InverterRun { ExternalAccessible := 'False'; ExternalVisible := 'False'; ExternalWritable := 'False'} : Bool;
      InverterReady { ExternalAccessible := 'False'; ExternalVisible := 'False'; ExternalWritable := 'False'} : Bool;
      HydrolockProtection { ExternalAccessible := 'False'; ExternalVisible := 'False'; ExternalWritable := 'False'} : Bool;
      A3400 { ExternalAccessible := 'False'; ExternalVisible := 'False'; ExternalWritable := 'False'; S7_SetPoint := 'False'} : "fbHMIEvent";
   END_VAR

   VAR_TEMP 
      PerformanceSetpointSelected : Real;   // [%] Selected performance setpoint
   END_VAR


BEGIN
	// Select motor setpoint and handle ready & run signals
	// NOTE: ramps are hardcoded, this is not ideal, should be in DB_CurrentSettings somewhere to make it easier to set up a new machine
	
	IF "DB_System".bEmergencyStop = TRUE THEN
	    #NEngineSetpoint := 0.0;
	ELSE
	    // Select setpoint
	    IF "DB_Regulators".PerformanceControl.ManualMode.ForcePowerSetpoint = TRUE THEN 
	        #PerformanceSetpointSelected := "DB_Regulators".PerformanceControl.ManualMode.ForcePowerSetpointValue;
	    ELSE
	        #PerformanceSetpointSelected := #"PerformanceSetpoint";
	    END_IF;
	
	    // Scale setpoint to RPM
	    #NEngineRequest := #PerformanceSetpointSelected / 100.0 * "DB_CurrentSetting".MissingSetting.Compressor.MaxOperationalSpeed;
	
	    // Limit setpoint
	    #NEngineRequest := LIMIT(IN := #NEngineRequest,
	                             MN := "DB_CurrentSetting".MissingSetting.Compressor.MinOperationalSpeed,
	                             MX := "DB_CurrentSetting".MissingSetting.Compressor.MaxOperationalSpeed);
	
	    CASE "DB_State".State.State_Number OF
	        0..1: // Init, offline modes
	            #NEngineSetpoint := 0.0;
	            #InverterReady := FALSE;
	            #InverterRun := FALSE;
	        2: // Standby
	            // If coming from one of the running modes, ramp down and stop
	            "RampLimiter"(InputValue            := 0.0,
	                          "PositivChange per_s" := 0.0,
	                          "NegativChange per_s" := -50.0,
	                          fCycleTime            := "DB_System".fCycleTime,
	                          OutputValue           := #NEngineSetpoint);
	            IF "DB_State".RunningConditions.CompressorStopped = TRUE THEN
	                #InverterReady := FALSE;
	                #InverterRun := FALSE;
	            END_IF;
	        3:  // PrepareStart
	            #NEngineSetpoint := 0.0;
	            #InverterReady := TRUE;
	        4:  // Start
	            IF "DB_State".RunningConditions.DoWarmStart = TRUE OR "DB_Regulators".PurgeControl.bDone = TRUE THEN
	                #InverterRun := TRUE;
	                // Preset the speed
	                #NEngineSetpoint := MAX(IN1 := #NEngineSetpoint, IN2 := "DB_CurrentSetting".MissingSetting.Compressor.MinStartupSpeed);   
	                "RampLimiter"(InputValue            := "DB_CurrentSetting".MissingSetting.System.HydrolockSpeed,                                  
	                              "PositivChange per_s" := 60.0,
	                              "NegativChange per_s" := -50.0,
	                              fCycleTime            := "DB_System".fCycleTime,
	                              OutputValue           := #NEngineSetpoint);
	            ELSE
	                // Note: Purge Control handles its own ramping
	                #NEngineSetpoint := "DB_Regulators".PurgeControl.fSpinOut;
	                #InverterRun := ("DB_Regulators".PurgeControl.nMode = 1);   // Don't touch
	            END_IF;
	
	            
	        5:  // Warmup
	            IF "DB_State".RunningConditions.RiskOfHydrolock = TRUE THEN
	                "RampLimiter"(InputValue            := MIN(IN1 := #NEngineSetpoint, IN2 := "DB_CurrentSetting".MissingSetting.System.HydrolockSpeed),
	                              "PositivChange per_s" := 0.0,
	                              "NegativChange per_s" := -500.0,
	                              fCycleTime            := "DB_System".fCycleTime,
	                              OutputValue           := #NEngineSetpoint);
	            ELSE
	                // Preset the speed
	                #NEngineSetpoint := MAX(IN1 := #NEngineSetpoint, IN2 := "DB_CurrentSetting".MissingSetting.Compressor.MinOperationalSpeed);
	                "RampLimiter"(InputValue := MIN(IN1 := "DB_CurrentSetting".MissingSetting.Compressor.WarmupSpeed, IN2 := #NEngineRequest),
	                              "PositivChange per_s" := 15.0,
	                              "NegativChange per_s" := -50.0,
	                              fCycleTime            := "DB_System".fCycleTime,
	                              OutputValue           := #NEngineSetpoint);
	            END_IF;
	        6:  // Running
	            IF "DB_State".RunningConditions.RiskOfHydrolock = TRUE THEN
	                "RampLimiter"(InputValue            := MIN(IN1 := #NEngineSetpoint, IN2 := "DB_CurrentSetting".MissingSetting.System.HydrolockSpeed),
	                              "PositivChange per_s" := 0.0,
	                              "NegativChange per_s" := -500.0,
	                              fCycleTime            := "DB_System".fCycleTime,
	                              OutputValue           := #NEngineSetpoint);
	            ELSE
	                "RampLimiter"(InputValue            := #NEngineRequest,
	                              "PositivChange per_s" := 30.0,
	                              "NegativChange per_s" := -30.0,
	                              fCycleTime            := "DB_System".fCycleTime,
	                              OutputValue           := #NEngineSetpoint);
	            END_IF;
	        7:  // Stopping
	            IF #FastStop = TRUE THEN
	                // Unconditional rampdown
	                "RampLimiter"(InputValue            := 0.0,
	                              "PositivChange per_s" := 0.0,
	                              "NegativChange per_s" := -500.0,
	                              fCycleTime            := "DB_System".fCycleTime,
	                              OutputValue           := #NEngineSetpoint);
	            ELSIF "DB_State".RunningConditions.SuctionLineDry = FALSE THEN
	                // Dry suction line at lower speed
	                "RampLimiter"(InputValue            := "DB_CurrentSetting".MissingSetting.Compressor.MinOperationalSpeed,
	                              "PositivChange per_s" := 60.0,
	                              "NegativChange per_s" := -50.0,
	                              fCycleTime            := "DB_System".fCycleTime,
	                              OutputValue           := #NEngineSetpoint);
	            ELSE
	                // Normal rampdown
	                "RampLimiter"(InputValue            := 0.0,
	                              "PositivChange per_s" := 0.0,
	                              "NegativChange per_s" := -50.0,
	                              fCycleTime            := "DB_System".fCycleTime,
	                              OutputValue           := #NEngineSetpoint);
	            END_IF;
	    END_CASE;
	
	END_IF;
	
	// Assign to inverter bits
	"DB_InverterDrives".HBL_SC_10.Cmd.bReady := #InverterReady;
	"DB_InverterDrives".HBL_SC_10.Cmd.bRun := #InverterRun;
	
END_FUNCTION_BLOCK

FUNCTION_BLOCK "ValveControl"   // FB27, FBD
TITLE = Setpoint selection & drivers
{ S7_Optimized_Access := 'TRUE' }
VERSION : 0.1
// stored: AutoNumber true, IsIECCheckEnabled false, IsRetainMemResEnabled false, MemoryReserve 100, SetENOAutomatically false, UDAEnableTagReadback false
   VAR_INPUT
      ValveSetpoint { ExternalAccessible := 'False'; ExternalVisible := 'False'; ExternalWritable := 'False'} : Real;   // [%] Valve position from regulator
   END_VAR
   VAR
      Setpoint { ExternalAccessible := 'False'; ExternalVisible := 'False'; ExternalWritable := 'False'} : Real;   // [%] Selected valve position
   END_VAR
   VAR_TEMP   // added for the SCL form of the ladder/FBD networks
      _w1 : Bool;
      _w2 : Bool;
   END_VAR
BEGIN

REGION Network 1 (SCL): Comment & history
   // Run valve drivers and do any switching of setpoints in case a valve is part of more than one control axis
END_REGION

REGION Network 2: Expansion valves
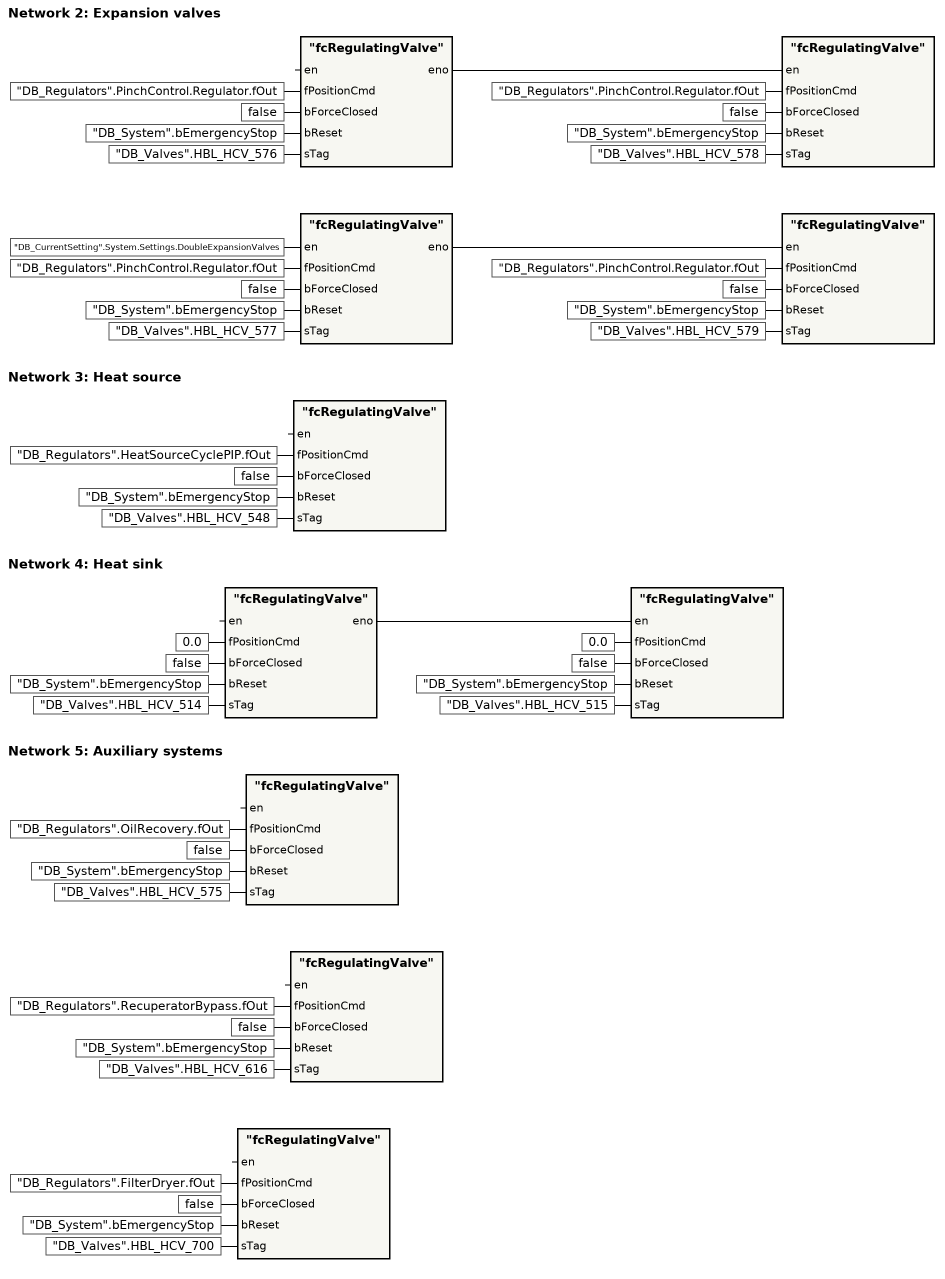
   "fcRegulatingValve"(fPositionCmd := "DB_Regulators".PinchControl.Regulator.fOut,
                       bForceClosed := false,
                       bReset := "DB_System".bEmergencyStop,
                       sTag := "DB_Valves".HBL_HCV_576,
                       ENO => #_w1);
   IF #_w1 THEN
       "fcRegulatingValve"(fPositionCmd := "DB_Regulators".PinchControl.Regulator.fOut,
                           bForceClosed := false,
                           bReset := "DB_System".bEmergencyStop,
                           sTag := "DB_Valves".HBL_HCV_578);
   END_IF;
   "fcRegulatingValve"(EN := "DB_CurrentSetting".System.Settings.DoubleExpansionValves,
                       fPositionCmd := "DB_Regulators".PinchControl.Regulator.fOut,
                       bForceClosed := false,
                       bReset := "DB_System".bEmergencyStop,
                       sTag := "DB_Valves".HBL_HCV_577,
                       ENO => #_w2);
   IF #_w2 THEN
       "fcRegulatingValve"(fPositionCmd := "DB_Regulators".PinchControl.Regulator.fOut,
                           bForceClosed := false,
                           bReset := "DB_System".bEmergencyStop,
                           sTag := "DB_Valves".HBL_HCV_579);
   END_IF;
END_REGION

REGION Network 3: Heat source
   "fcRegulatingValve"(fPositionCmd := "DB_Regulators".HeatSourceCyclePIP.fOut,
                       bForceClosed := false,
                       bReset := "DB_System".bEmergencyStop,
                       sTag := "DB_Valves".HBL_HCV_548);
END_REGION

REGION Network 4: Heat sink
   "fcRegulatingValve"(fPositionCmd := 0.0,
                       bForceClosed := false,
                       bReset := "DB_System".bEmergencyStop,
                       sTag := "DB_Valves".HBL_HCV_514,
                       ENO => #_w1);
   IF #_w1 THEN
       "fcRegulatingValve"(fPositionCmd := 0.0,
                           bForceClosed := false,
                           bReset := "DB_System".bEmergencyStop,
                           sTag := "DB_Valves".HBL_HCV_515);
   END_IF;
END_REGION

REGION Network 5: Auxiliary systems
   "fcRegulatingValve"(fPositionCmd := "DB_Regulators".OilRecovery.fOut,
                       bForceClosed := false,
                       bReset := "DB_System".bEmergencyStop,
                       sTag := "DB_Valves".HBL_HCV_575);
   "fcRegulatingValve"(fPositionCmd := "DB_Regulators".RecuperatorBypass.fOut,
                       bForceClosed := false,
                       bReset := "DB_System".bEmergencyStop,
                       sTag := "DB_Valves".HBL_HCV_616);
   "fcRegulatingValve"(fPositionCmd := "DB_Regulators".FilterDryer.fOut,
                       bForceClosed := false,
                       bReset := "DB_System".bEmergencyStop,
                       sTag := "DB_Valves".HBL_HCV_700);
END_REGION
END_FUNCTION_BLOCK

FUNCTION_BLOCK "fbSafetyRelay"
{ S7_Optimized_Access := 'TRUE' }
VERSION : 0.1
   VAR_INPUT 
      bStatus : Bool;   // Safety relay status 1 = ok, 0 = E-stop
   END_VAR

   VAR_OUTPUT 
      bExternalEstop : Bool;   // External E-stop is active
      bResetFailed : Bool;   // Failed to reset safety relay
   END_VAR

   VAR_IN_OUT 
      sTag : "stSafetyRelay";
   END_VAR

   VAR 
      SequenceTimer {InstructionName := 'TON_TIME'; LibVersion := '1.0'; S7_SetPoint := 'False'} : TON_TIME;
      ResetTimeout {InstructionName := 'TON_TIME'; LibVersion := '1.0'} : TON_TIME;
      ResetReq {InstructionName := 'R_TRIG'; LibVersion := '1.0'} : R_TRIG;   // Make sure command is an edge
   END_VAR


BEGIN
	// Sequencer to reset the safety relay.
	// 1. Close the PLC's E-stop loop output relay
	// 2. Send the reset command to the Safety relay
	// 3. Wait for a positive response, give up after timeout
	
	// Copy status into tag
	#sTag.bStatus := #bStatus;
	
	// Make reset signal an edge to prevent endless retriggering
	#ResetReq(CLK := #sTag.bResetReq);
	
	// Evaluate timers outside state machine so they reset properly
	#SequenceTimer(IN := (#sTag.nState = 1), PT := #sTag.tResetLoopTime);
	#ResetTimeout(IN := (#sTag.nState = 2), PT := #sTag.tResetTimeout);
	
	// Safety relay reset cycle
	CASE #sTag.nState OF
	    0: // Safety relay is tripped/open
	        IF #ResetReq.Q = TRUE THEN
	            #sTag.bResetLoop := TRUE;
	            #sTag.nState := 1;
	            #sTag.bResetFailed := FALSE;
	        ELSIF #bStatus = TRUE THEN
	            // Externally reset
	            #sTag.bResetFailed := FALSE;
	            #sTag.nState := 3;
	        END_IF;
	    1: // Give loop relay time to close
	        IF #SequenceTimer.Q = TRUE THEN 
	            #sTag.bResetCmd := TRUE;
	            #sTag.nState := 2;
	        END_IF;
	    2: // Wait for safety relay feedback or timeout
	        IF #bStatus = TRUE THEN
	            #sTag.bResetLoop := FALSE;
	            #sTag.bResetCmd := FALSE;
	            #sTag.nState := 3;
	        ELSIF #ResetTimeout.Q = TRUE THEN
	            #sTag.bResetLoop := FALSE;
	            #sTag.bResetCmd := FALSE;
	            #sTag.bResetFailed := TRUE;
	            #sTag.nState := 0;
	        END_IF;
	    3: // Safety relay is closed
	        IF #bStatus = FALSE THEN
	            #sTag.nState := 0;
	        END_IF;
	END_CASE;
	
	// Local outputs
	#bExternalEstop := NOT #bStatus;
	#bResetFailed := #sTag.bResetFailed;
	
END_FUNCTION_BLOCK

FUNCTION_BLOCK "StartStopControl"   // FB30, FBD
{ S7_Optimized_Access := 'TRUE' }
VERSION : 0.1
// stored: AutoNumber true, IsIECCheckEnabled false, IsRetainMemResEnabled false, MemoryReserve 0, SetENOAutomatically false, UDAEnableTagReadback false
   VAR_OUTPUT
      Run : Bool;   // 1 = run, 0 = stop
   END_VAR
   VAR
      StartRequestHMI { ExternalAccessible := 'False'; ExternalVisible := 'False'; ExternalWritable := 'False'; S7_SetPoint := 'True'} : R_TRIG;
      StartRequestApplication { ExternalAccessible := 'False'; ExternalVisible := 'False'; ExternalWritable := 'False'; S7_SetPoint := 'True'} : R_TRIG;
      StopRequestHMI { ExternalAccessible := 'False'; ExternalVisible := 'False'; ExternalWritable := 'False'; S7_SetPoint := 'True'} : R_TRIG;
      StopRequestApplication { ExternalAccessible := 'False'; ExternalVisible := 'False'; ExternalWritable := 'False'; S7_SetPoint := 'True'} : R_TRIG;
      EmergencyStopWaitTime { S7_SetPoint := 'True'} : TOF_TIME;
      StopRequestCriticalAlarm { S7_SetPoint := 'True'} : Bool;
   END_VAR
   VAR_TEMP
      StopRequestRegulatorFault : Bool;
   END_VAR
BEGIN

REGION Network 1: Start request signals
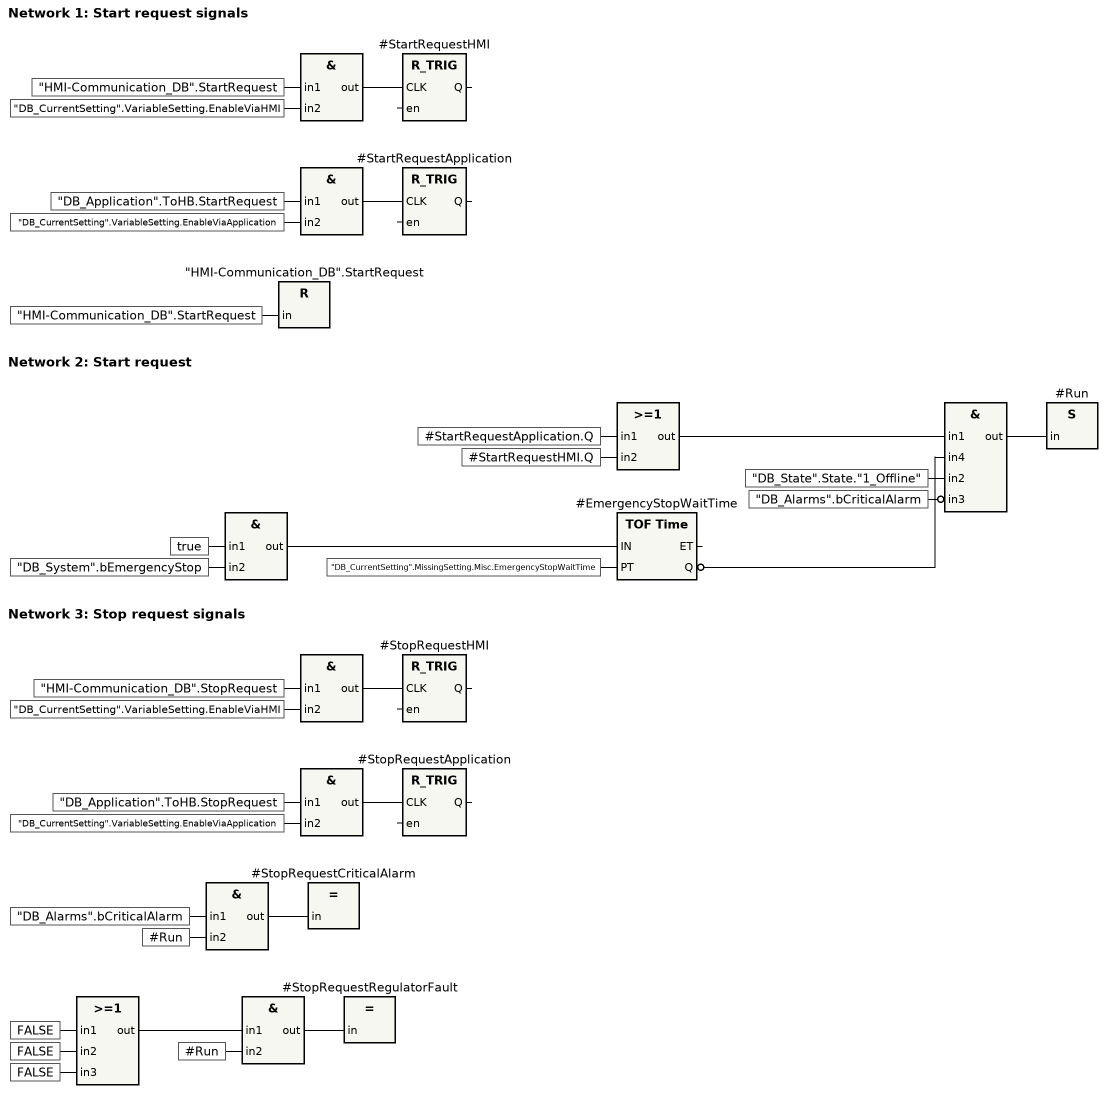
   #StartRequestHMI(CLK := "HMI-Communication_DB".StartRequest AND "DB_CurrentSetting".VariableSetting.EnableViaHMI);   // R_TRIG
   #StartRequestApplication(CLK := "DB_Application".ToHB.StartRequest AND "DB_CurrentSetting".VariableSetting.EnableViaApplication);   // R_TRIG
   IF "HMI-Communication_DB".StartRequest THEN "HMI-Communication_DB".StartRequest := FALSE; END_IF;
END_REGION

REGION Network 2: Start request
   // Start conditions:
   // 1. Start request from one of the control sources
   // 2. State 1 
   // 3. No critical alarms active
   // 4. E-stop lockout timer has expired
   // Also reset alarms
   #EmergencyStopWaitTime(IN := true AND "DB_System".bEmergencyStop,   // TOF
                          PT := "DB_CurrentSetting".MissingSetting.Misc.EmergencyStopWaitTime);
   IF (#StartRequestApplication.Q OR #StartRequestHMI.Q) AND NOT #EmergencyStopWaitTime.Q AND "DB_State".State."1_Offline" AND NOT "DB_Alarms".bCriticalAlarm THEN
       #Run := TRUE;
   END_IF;
END_REGION

REGION Network 3: Stop request signals
   // ##FIX decide what to do about regulator faults.
   #StopRequestHMI(CLK := "HMI-Communication_DB".StopRequest AND "DB_CurrentSetting".VariableSetting.EnableViaHMI);   // R_TRIG
   #StopRequestApplication(CLK := "DB_Application".ToHB.StopRequest AND "DB_CurrentSetting".VariableSetting.EnableViaApplication);   // R_TRIG
   #StopRequestCriticalAlarm := "DB_Alarms".bCriticalAlarm AND #Run;
   #StopRequestRegulatorFault := (FALSE OR FALSE OR FALSE) AND #Run;
END_REGION

REGION Network 4: Stop request
   // Stop condition is one of:
   // 1. Stop request from one of the control sources (HMI or App PLC)
   // 2. Forced into State 7 Stop (and the machine should follow)
   // 3. Critical Alarm
   // 4. Emergency Stop. (This is also technically a critical alarm but alarms can be disabled)
   // 5. Regulator fault
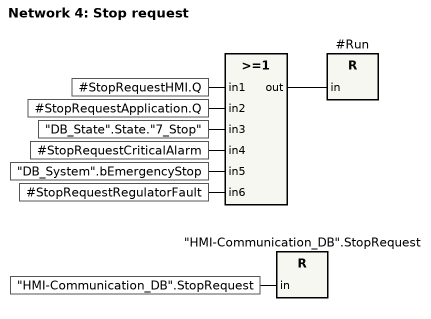
   IF #StopRequestHMI.Q OR #StopRequestApplication.Q OR "DB_State".State."7_Stop" OR #StopRequestCriticalAlarm OR "DB_System".bEmergencyStop OR #StopRequestRegulatorFault THEN
       #Run := FALSE;
   END_IF;
   IF "HMI-Communication_DB".StopRequest THEN "HMI-Communication_DB".StopRequest := FALSE; END_IF;
END_REGION
END_FUNCTION_BLOCK

FUNCTION_BLOCK "OutputProcessing"   // FB11, FBD
TITLE = Output mapping
{ S7_Optimized_Access := 'TRUE' }
VERSION : 0.1
// stored: AutoNumber true, IsIECCheckEnabled false, IsRetainMemResEnabled false, MemoryReserve 0, SetENOAutomatically false, UDAEnableTagReadback false
BEGIN

REGION Network 1: Digital
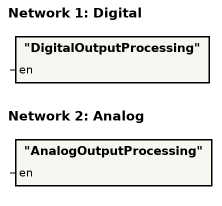
   "DigitalOutputProcessing"();
END_REGION

REGION Network 2: Analog
   "AnalogOutputProcessing"();
END_REGION
END_FUNCTION_BLOCK

FUNCTION "DigitalOutputProcessing" : Void   // FC11, FBD
TITLE = Output mapping
{ S7_Optimized_Access := 'TRUE' }
VERSION : 0.1
// stored: AutoNumber true, IsIECCheckEnabled false, SetENOAutomatically false, UDAEnableTagReadback false
   VAR_TEMP
      Spare : Bool;
   END_VAR
BEGIN

REGION Network 1: Emergency Stop output
   // 1 = ok, 0 = emergency stop
   // If emergency stop is not active, or you want to reset the safety relay, output is high.
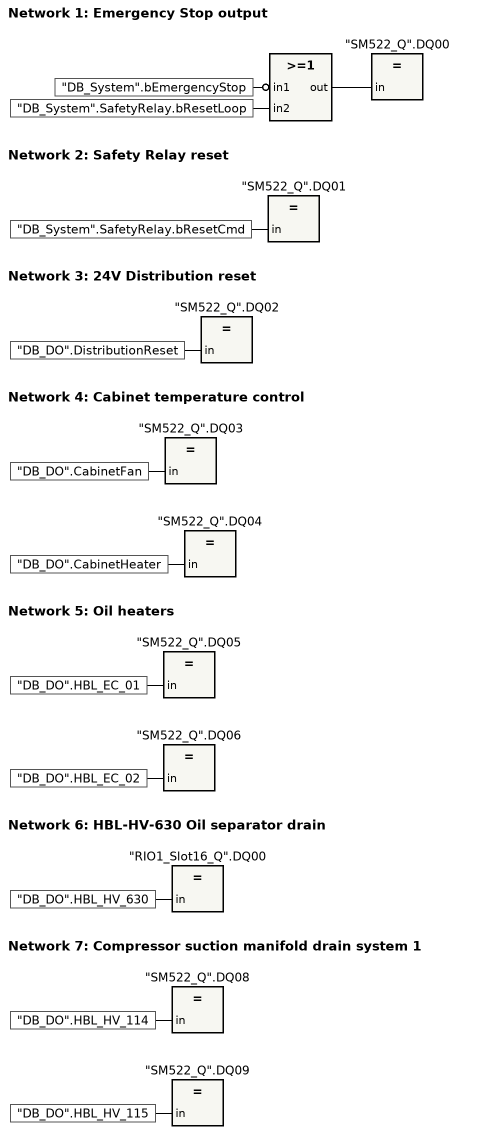
   "SM522_Q".DQ00 := NOT "DB_System".bEmergencyStop OR "DB_System".SafetyRelay.bResetLoop;
END_REGION

REGION Network 2: Safety Relay reset
   "SM522_Q".DQ01 := "DB_System".SafetyRelay.bResetCmd;
END_REGION

REGION Network 3: 24V Distribution reset
   "SM522_Q".DQ02 := "DB_DO".DistributionReset;
END_REGION

REGION Network 4: Cabinet temperature control
   "SM522_Q".DQ03 := "DB_DO".CabinetFan;
   "SM522_Q".DQ04 := "DB_DO".CabinetHeater;
END_REGION

REGION Network 5: Oil heaters
   "SM522_Q".DQ05 := "DB_DO".HBL_EC_01;
   "SM522_Q".DQ06 := "DB_DO".HBL_EC_02;
END_REGION

REGION Network 6: HBL-HV-630 Oil separator drain
   "RIO1_Slot16_Q".DQ00 := "DB_DO".HBL_HV_630;
END_REGION

REGION Network 7: Compressor suction manifold drain system 1
   // Valves directly from suction manifold to sump (optional)
   "SM522_Q".DQ08 := "DB_DO".HBL_HV_114;
   "SM522_Q".DQ09 := "DB_DO".HBL_HV_115;
END_REGION

REGION Network 8: Shaft Seal Cartridge (SSC)
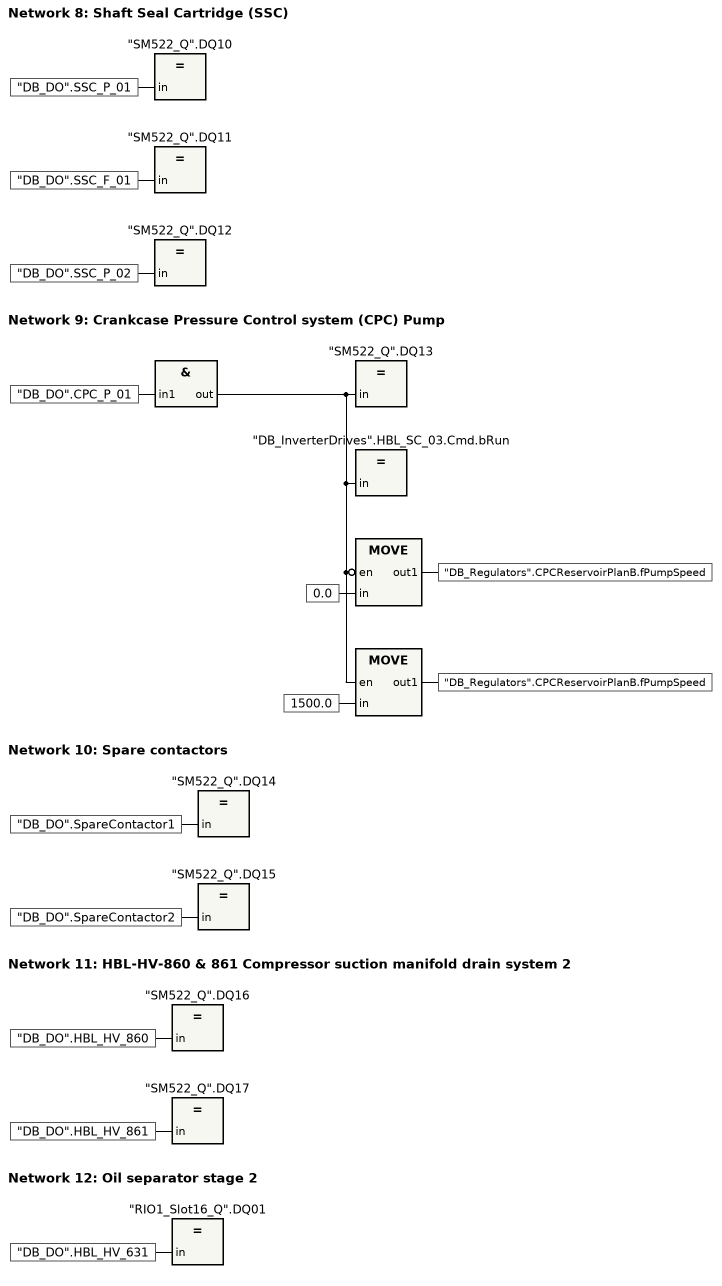
   "SM522_Q".DQ10 := "DB_DO".SSC_P_01;
   "SM522_Q".DQ11 := "DB_DO".SSC_F_01;
   "SM522_Q".DQ12 := "DB_DO".SSC_P_02;
END_REGION

REGION Network 9: Crankcase Pressure Control system (CPC) Pump
   // 10.02.2025 TSS: Normally DQ13, but now an inverter. And this is the ugly hack to make it work until we know how it really should be.
   "SM522_Q".DQ13 := "DB_DO".CPC_P_01;
   "DB_InverterDrives".HBL_SC_03.Cmd.bRun := "DB_DO".CPC_P_01;
   IF NOT "DB_DO".CPC_P_01 THEN "DB_Regulators".CPCReservoirPlanB.fPumpSpeed := 0.0; END_IF;
   IF "DB_DO".CPC_P_01 THEN "DB_Regulators".CPCReservoirPlanB.fPumpSpeed := 1500.0; END_IF;
END_REGION

REGION Network 10: Spare contactors
   "SM522_Q".DQ14 := "DB_DO".SpareContactor1;
   "SM522_Q".DQ15 := "DB_DO".SpareContactor2;
END_REGION

REGION Network 11: HBL-HV-860 & 861 Compressor suction manifold drain system 2
   // Valves to share the CPC system with the Purge controller
   "SM522_Q".DQ16 := "DB_DO".HBL_HV_860;
   "SM522_Q".DQ17 := "DB_DO".HBL_HV_861;
END_REGION

REGION Network 12: Oil separator stage 2
   "RIO1_Slot16_Q".DQ01 := "DB_DO".HBL_HV_631;
END_REGION

REGION Network 13: HBL-HV-640
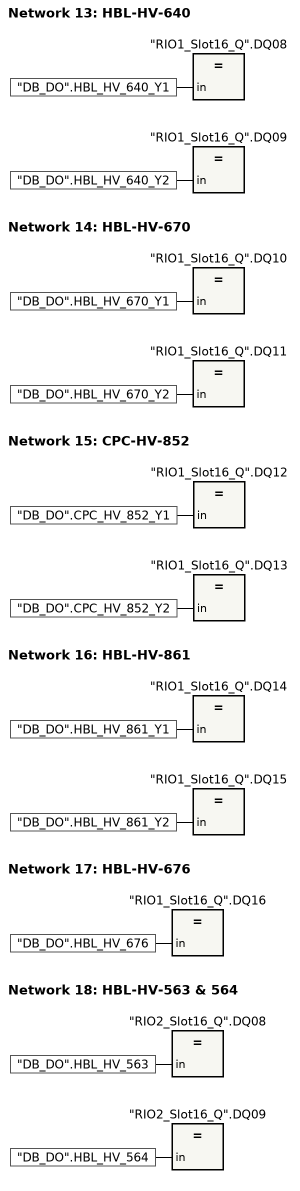
   "RIO1_Slot16_Q".DQ08 := "DB_DO".HBL_HV_640_Y1;
   "RIO1_Slot16_Q".DQ09 := "DB_DO".HBL_HV_640_Y2;
END_REGION

REGION Network 14: HBL-HV-670
   "RIO1_Slot16_Q".DQ10 := "DB_DO".HBL_HV_670_Y1;
   "RIO1_Slot16_Q".DQ11 := "DB_DO".HBL_HV_670_Y2;
END_REGION

REGION Network 15: CPC-HV-852
   "RIO1_Slot16_Q".DQ12 := "DB_DO".CPC_HV_852_Y1;
   "RIO1_Slot16_Q".DQ13 := "DB_DO".CPC_HV_852_Y2;
END_REGION

REGION Network 16: HBL-HV-861
   "RIO1_Slot16_Q".DQ14 := "DB_DO".HBL_HV_861_Y1;
   "RIO1_Slot16_Q".DQ15 := "DB_DO".HBL_HV_861_Y2;
END_REGION

REGION Network 17: HBL-HV-676
   "RIO1_Slot16_Q".DQ16 := "DB_DO".HBL_HV_676;
END_REGION

REGION Network 18: HBL-HV-563 & 564
   "RIO2_Slot16_Q".DQ08 := "DB_DO".HBL_HV_563;
   "RIO2_Slot16_Q".DQ09 := "DB_DO".HBL_HV_564;
END_REGION
END_FUNCTION

FUNCTION "AnalogOutputProcessing" : Void   // FC12, FBD
TITLE = Output mapping and scaling
{ S7_Optimized_Access := 'TRUE' }
VERSION : 0.1
// stored: AutoNumber true, IsIECCheckEnabled false, SetENOAutomatically false, UDAEnableTagReadback false
BEGIN

REGION Network 1: HBL-HCV-576
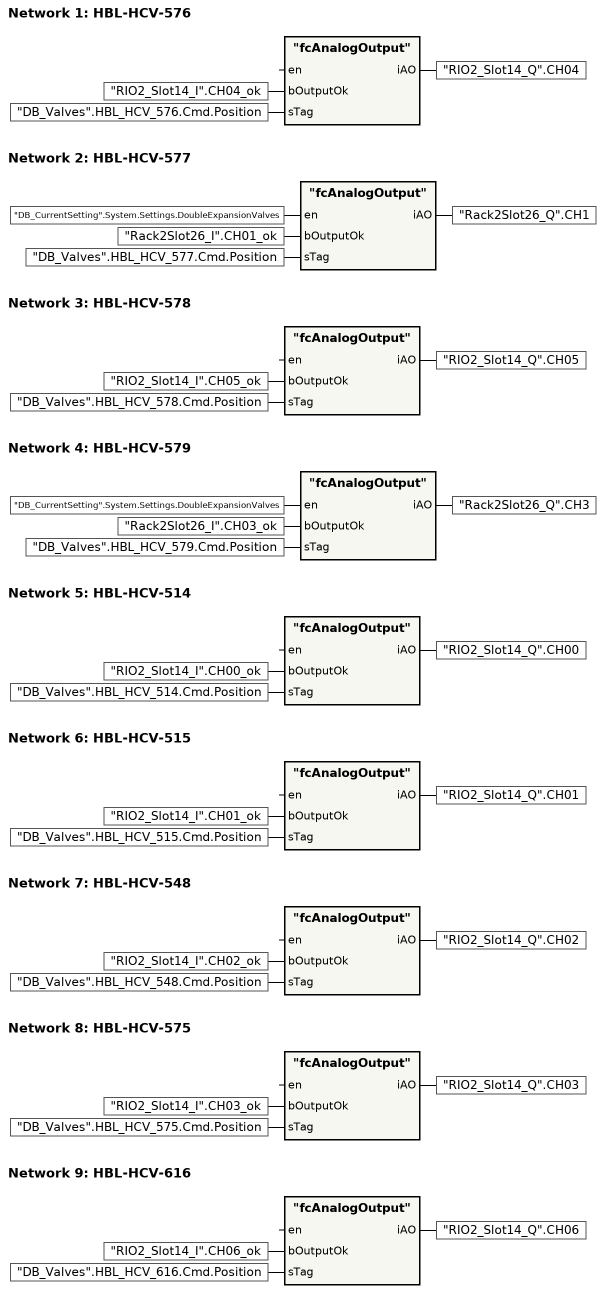
   "fcAnalogOutput"(bOutputOk := "RIO2_Slot14_I".CH04_ok,
                    sTag := "DB_Valves".HBL_HCV_576.Cmd.Position,
                    iAO => "RIO2_Slot14_Q".CH04);
END_REGION

REGION Network 2: HBL-HCV-577
   IF "DB_CurrentSetting".System.Settings.DoubleExpansionValves THEN
       "fcAnalogOutput"(bOutputOk := "Rack2Slot26_I".CH01_ok,
                        sTag := "DB_Valves".HBL_HCV_577.Cmd.Position,
                        iAO => "Rack2Slot26_Q".CH1);
   END_IF;
END_REGION

REGION Network 3: HBL-HCV-578
   "fcAnalogOutput"(bOutputOk := "RIO2_Slot14_I".CH05_ok,
                    sTag := "DB_Valves".HBL_HCV_578.Cmd.Position,
                    iAO => "RIO2_Slot14_Q".CH05);
END_REGION

REGION Network 4: HBL-HCV-579
   IF "DB_CurrentSetting".System.Settings.DoubleExpansionValves THEN
       "fcAnalogOutput"(bOutputOk := "Rack2Slot26_I".CH03_ok,
                        sTag := "DB_Valves".HBL_HCV_579.Cmd.Position,
                        iAO => "Rack2Slot26_Q".CH3);
   END_IF;
END_REGION

REGION Network 5: HBL-HCV-514
   "fcAnalogOutput"(bOutputOk := "RIO2_Slot14_I".CH00_ok,
                    sTag := "DB_Valves".HBL_HCV_514.Cmd.Position,
                    iAO => "RIO2_Slot14_Q".CH00);
END_REGION

REGION Network 6: HBL-HCV-515
   "fcAnalogOutput"(bOutputOk := "RIO2_Slot14_I".CH01_ok,
                    sTag := "DB_Valves".HBL_HCV_515.Cmd.Position,
                    iAO => "RIO2_Slot14_Q".CH01);
END_REGION

REGION Network 7: HBL-HCV-548
   "fcAnalogOutput"(bOutputOk := "RIO2_Slot14_I".CH02_ok,
                    sTag := "DB_Valves".HBL_HCV_548.Cmd.Position,
                    iAO => "RIO2_Slot14_Q".CH02);
END_REGION

REGION Network 8: HBL-HCV-575
   "fcAnalogOutput"(bOutputOk := "RIO2_Slot14_I".CH03_ok,
                    sTag := "DB_Valves".HBL_HCV_575.Cmd.Position,
                    iAO => "RIO2_Slot14_Q".CH03);
END_REGION

REGION Network 9: HBL-HCV-616
   "fcAnalogOutput"(bOutputOk := "RIO2_Slot14_I".CH06_ok,
                    sTag := "DB_Valves".HBL_HCV_616.Cmd.Position,
                    iAO => "RIO2_Slot14_Q".CH06);
END_REGION

REGION Network 10: HBL-HCV-700
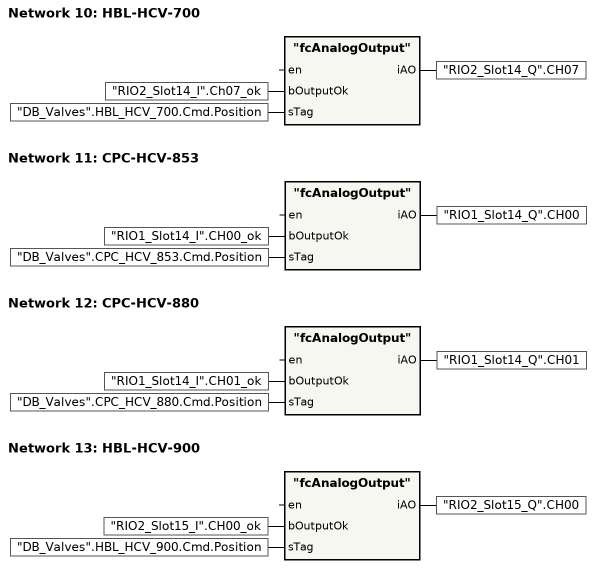
   "fcAnalogOutput"(bOutputOk := "RIO2_Slot14_I".Ch07_ok,
                    sTag := "DB_Valves".HBL_HCV_700.Cmd.Position,
                    iAO => "RIO2_Slot14_Q".CH07);
END_REGION

REGION Network 11: CPC-HCV-853
   "fcAnalogOutput"(bOutputOk := "RIO1_Slot14_I".CH00_ok,
                    sTag := "DB_Valves".CPC_HCV_853.Cmd.Position,
                    iAO => "RIO1_Slot14_Q".CH00);
END_REGION

REGION Network 12: CPC-HCV-880
   "fcAnalogOutput"(bOutputOk := "RIO1_Slot14_I".CH01_ok,
                    sTag := "DB_Valves".CPC_HCV_880.Cmd.Position,
                    iAO => "RIO1_Slot14_Q".CH01);
END_REGION

REGION Network 13: HBL-HCV-900
   "fcAnalogOutput"(bOutputOk := "RIO2_Slot15_I".CH00_ok,
                    sTag := "DB_Valves".HBL_HCV_900.Cmd.Position,
                    iAO => "RIO2_Slot15_Q".CH00);
END_REGION
END_FUNCTION

FUNCTION_BLOCK "Diagnosis"   // FB1, FBD
TITLE = Misc alarm handling
{ S7_Optimized_Access := 'TRUE' }
VERSION : 0.1
// stored: AutoNumber true, IsIECCheckEnabled false, IsRetainMemResEnabled false, MemoryReserve 0, SetENOAutomatically false, UDAEnableTagReadback false
   VAR
      A0001 { ExternalAccessible := 'False'; ExternalVisible := 'False'; ExternalWritable := 'False'} : "fbHMIEvent";
      A1002 { ExternalAccessible := 'False'; ExternalVisible := 'False'; ExternalWritable := 'False'; S7_SetPoint := 'True'} : "fbHMIEvent";
      A1003 { ExternalAccessible := 'False'; ExternalVisible := 'False'; ExternalWritable := 'False'; S7_SetPoint := 'True'} : "fbHMIEvent";
   END_VAR
BEGIN

REGION Network 1: 0001 Watchdog timeout OB1
   // "DB_Alarms"."0001_WatchdogTimeoutOB1".bInput is written by OB80, but alarm is processed here (OB80 is not cyclic)
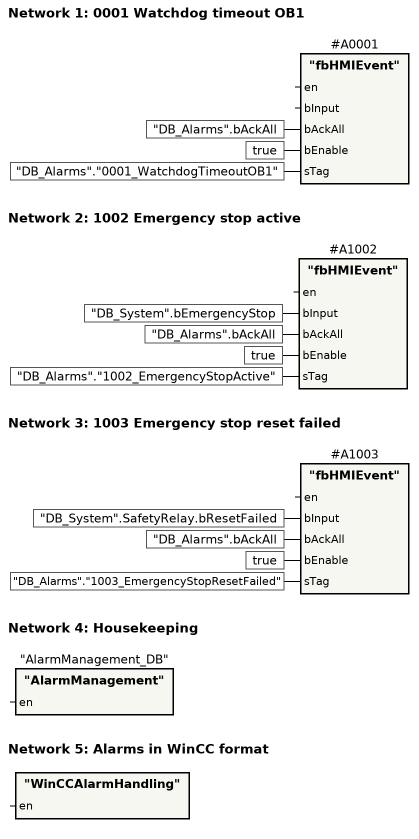
   #A0001(bAckAll := "DB_Alarms".bAckAll, bEnable := true, sTag := "DB_Alarms"."0001_WatchdogTimeoutOB1");   // "fbHMIEvent"
END_REGION

REGION Network 2: 1002 Emergency stop active
   #A1002(bInput := "DB_System".bEmergencyStop,   // "fbHMIEvent"
          bAckAll := "DB_Alarms".bAckAll,
          bEnable := true,
          sTag := "DB_Alarms"."1002_EmergencyStopActive");
END_REGION

REGION Network 3: 1003 Emergency stop reset failed
   #A1003(bInput := "DB_System".SafetyRelay.bResetFailed,   // "fbHMIEvent"
          bAckAll := "DB_Alarms".bAckAll,
          bEnable := true,
          sTag := "DB_Alarms"."1003_EmergencyStopResetFailed");
END_REGION

REGION Network 4: Housekeeping
   "AlarmManagement_DB"();   // "AlarmManagement"
END_REGION

REGION Network 5: Alarms in WinCC format
   "WinCCAlarmHandling"();
END_REGION

REGION Network 6 (SCL): Alarms to App PLC - Group 0 & 1
   // Group 0-System
   "DB_Application".FromHB.Alarms[0] := "DB_WinCCAlarms"."0-System"."0001_WatchdogTimeoutOB1".Memory.%X0;
   "DB_Application".FromHB.Alarms[1] := "DB_WinCCAlarms"."0-System"."0003_InitCurrenSettingsFailed".Memory.%X0;
   "DB_Application".FromHB.Alarms[2] := "DB_WinCCAlarms"."0-System"."0006_CPUinErrorState".Memory.%X0;

   // Group 1-IO
   "DB_Application".FromHB.Alarms[3]  := "DB_WinCCAlarms"."1-IO"."1001_ConnectionToWinCClost".Memory.%X0;
   "DB_Application".FromHB.Alarms[4]  := "DB_WinCCAlarms"."1-IO"."1002_EmergencyStopActive".Memory.%X0;
   "DB_Application".FromHB.Alarms[5]  := "DB_WinCCAlarms"."1-IO"."1003_SafetyRelayResetFailed".Memory.%X0;
   "DB_Application".FromHB.Alarms[6]  := "DB_WinCCAlarms"."1-IO"."1004_HBL_PS_01_X2".Memory.%X0;
   "DB_Application".FromHB.Alarms[7]  := "DB_WinCCAlarms"."1-IO"."1101_HBL_SC_01_CommError".Memory.%X0;
   "DB_Application".FromHB.Alarms[8]  := "DB_WinCCAlarms"."1-IO"."1102_HBL_SC_02_CommError".Memory.%X0;
   "DB_Application".FromHB.Alarms[9]  := "DB_WinCCAlarms"."1-IO"."1110_HBL_SC_10_CommError".Memory.%X0;
   "DB_Application".FromHB.Alarms[10] := "DB_WinCCAlarms"."1-IO"."1121_HBL_SC_01_Tripped".Memory.%X0;
   "DB_Application".FromHB.Alarms[11] := "DB_WinCCAlarms"."1-IO"."1122_HBL_SC_02_Tripped".Memory.%X0;
   "DB_Application".FromHB.Alarms[12] := "DB_WinCCAlarms"."1-IO"."1130_HBL_SC_10_Tripped".Memory.%X0;
   "DB_Application".FromHB.Alarms[13] := "DB_WinCCAlarms"."1-IO"."1140_HBL_SC_01_RunFailure".Memory.%X0;
   "DB_Application".FromHB.Alarms[14] := "DB_WinCCAlarms"."1-IO"."1142_HBL_SC_02_RunFailure".Memory.%X0;
   "DB_Application".FromHB.Alarms[15] := "DB_WinCCAlarms"."1-IO"."1150_HBL_SC_10_RunFailure".Memory.%X0;

   "DB_Application".FromHB.Alarms[16] := "DB_WinCCAlarms"."1-IO"."1201_HBL_PT_01_Fault".Memory.%X0;
   "DB_Application".FromHB.Alarms[17] := "DB_WinCCAlarms"."1-IO"."1202_HBL_PT_02_Fault".Memory.%X0;
   "DB_Application".FromHB.Alarms[18] := "DB_WinCCAlarms"."1-IO"."1203_HBL_PT_03_Fault".Memory.%X0;
   "DB_Application".FromHB.Alarms[19] := "DB_WinCCAlarms"."1-IO"."1204_HBL_PT_04_Fault".Memory.%X0;
   "DB_Application".FromHB.Alarms[20] := "DB_WinCCAlarms"."1-IO"."1205_HBL_TT_05_Fault".Memory.%X0;
   "DB_Application".FromHB.Alarms[21] := "DB_WinCCAlarms"."1-IO"."1206_HBL_TT_06_Fault".Memory.%X0;
   "DB_Application".FromHB.Alarms[22] := "DB_WinCCAlarms"."1-IO"."1207_HBL_TT_07_Fault".Memory.%X0;
   "DB_Application".FromHB.Alarms[23] := "DB_WinCCAlarms"."1-IO"."1208_HBL_TT_08_Fault".Memory.%X0;
   "DB_Application".FromHB.Alarms[24] := "DB_WinCCAlarms"."1-IO"."1209_HBL_HCV_01_A1_Fault".Memory.%X0;
   "DB_Application".FromHB.Alarms[25] := "DB_WinCCAlarms"."1-IO"."1210_HBL_TT_10_Fault".Memory.%X0;
   "DB_Application".FromHB.Alarms[26] := "DB_WinCCAlarms"."1-IO"."1212_HBL_TT_12_Fault".Memory.%X0;
   "DB_Application".FromHB.Alarms[27] := "DB_WinCCAlarms"."1-IO"."1213_HBL_TT_13_Fault".Memory.%X0;
   "DB_Application".FromHB.Alarms[28] := "DB_WinCCAlarms"."1-IO"."1214_HBL_TT_14_Fault".Memory.%X0;
   "DB_Application".FromHB.Alarms[29] := "DB_WinCCAlarms"."1-IO"."1215_HBL_TT_15_Fault".Memory.%X0;
   "DB_Application".FromHB.Alarms[30] := "DB_WinCCAlarms"."1-IO"."1216_HBL_TT_16_Fault".Memory.%X0;
   "DB_Application".FromHB.Alarms[31] := "DB_WinCCAlarms"."1-IO"."1217_HBL_TT_17_Fault".Memory.%X0;
   "DB_Application".FromHB.Alarms[32] := "DB_WinCCAlarms"."1-IO"."1218_HBL_TT_18_Fault".Memory.%X0;
   "DB_Application".FromHB.Alarms[33] := "DB_WinCCAlarms"."1-IO"."1220_HBL_PT_960_Fault".Memory.%X0;
   "DB_Application".FromHB.Alarms[34] := "DB_WinCCAlarms"."1-IO"."1221_HBL_PT_05_Fault".Memory.%X0;
   "DB_Application".FromHB.Alarms[35] := "DB_WinCCAlarms"."1-IO"."1223_HBL_TT_03_Fault".Memory.%X0;
   "DB_Application".FromHB.Alarms[36] := "DB_WinCCAlarms"."1-IO"."1224_HBL_TT_23_Fault".Memory.%X0;
   "DB_Application".FromHB.Alarms[37] := "DB_WinCCAlarms"."1-IO"."1225_HBL_TT_24_Fault".Memory.%X0;
   "DB_Application".FromHB.Alarms[38] := "DB_WinCCAlarms"."1-IO"."1226_HBL_TT_25_Fault".Memory.%X0;
   "DB_Application".FromHB.Alarms[39] := "DB_WinCCAlarms"."1-IO"."1227_HBL_LT_01_Fault".Memory.%X0;
   "DB_Application".FromHB.Alarms[40] := "DB_WinCCAlarms"."1-IO"."1228_HBL_TT_21_Fault".Memory.%X0;
   "DB_Application".FromHB.Alarms[41] := "DB_WinCCAlarms"."1-IO"."1229_HBL_TT_22_Fault".Memory.%X0;
   "DB_Application".FromHB.Alarms[42] := "DB_WinCCAlarms"."1-IO"."1230_HBL_LT_02_Fault".Memory.%X0;
   "DB_Application".FromHB.Alarms[43] := "DB_WinCCAlarms"."1-IO"."1231_HBL_HCV_02_A1_Fault".Memory.%X0;
   "DB_Application".FromHB.Alarms[44] := "DB_WinCCAlarms"."1-IO"."1232_HBL_PT_13_Fault".Memory.%X0;
   "DB_Application".FromHB.Alarms[45] := "DB_WinCCAlarms"."1-IO"."1233_HBL_TT_20_Fault".Memory.%X0;
   "DB_Application".FromHB.Alarms[46] := "DB_WinCCAlarms"."1-IO"."1234_HBL_PT_14_Fault".Memory.%X0;
   "DB_Application".FromHB.Alarms[47] := "DB_WinCCAlarms"."1-IO"."1235_HBL_PT_18_Fault".Memory.%X0;
   "DB_Application".FromHB.Alarms[48] := "DB_WinCCAlarms"."1-IO"."1236_HBL_PT_19_Fault".Memory.%X0;
   "DB_Application".FromHB.Alarms[49] := "DB_WinCCAlarms"."1-IO"."1237_HBL_PT_25_Fault".Memory.%X0;
   "DB_Application".FromHB.Alarms[50] := "DB_WinCCAlarms"."1-IO"."1238_HBL_TT_31_Fault".Memory.%X0;
   "DB_Application".FromHB.Alarms[51] := "DB_WinCCAlarms"."1-IO"."1239_HBL_TT_33_Fault".Memory.%X0;
   "DB_Application".FromHB.Alarms[52] := "DB_WinCCAlarms"."1-IO"."1240_HBL_TT_35_Fault".Memory.%X0;
   "DB_Application".FromHB.Alarms[53] := "DB_WinCCAlarms"."1-IO"."1241_HBL_HCV_01_Fault".Memory.%X0;
   "DB_Application".FromHB.Alarms[54] := "DB_WinCCAlarms"."1-IO"."1242_HBL_HCV_02_Fault".Memory.%X0;
   "DB_Application".FromHB.Alarms[55] := "DB_WinCCAlarms"."1-IO"."1243_HBL_PT_07_Fault".Memory.%X0;
   "DB_Application".FromHB.Alarms[56] := "DB_WinCCAlarms"."1-IO"."1244_HBL_PT_08_Fault".Memory.%X0;
   "DB_Application".FromHB.Alarms[57] := "DB_WinCCAlarms"."1-IO"."1245_HBL_PT_09_Fault".Memory.%X0;
   "DB_Application".FromHB.Alarms[58] := "DB_WinCCAlarms"."1-IO"."1246_HBL_PT_10_Fault".Memory.%X0;
   "DB_Application".FromHB.Alarms[59] := "DB_WinCCAlarms"."1-IO"."1247_HBL_PT_11_Fault".Memory.%X0;
   "DB_Application".FromHB.Alarms[60] := "DB_WinCCAlarms"."1-IO"."1248_HBL_PT_12_Fault".Memory.%X0;
   "DB_Application".FromHB.Alarms[61] := "DB_WinCCAlarms"."1-IO"."1249_HBL_PT_15_Fault".Memory.%X0;
   "DB_Application".FromHB.Alarms[62] := FALSE;
   "DB_Application".FromHB.Alarms[63] := "DB_WinCCAlarms"."1-IO"."1251_HBL_PT_24_Fault".Memory.%X0;
   "DB_Application".FromHB.Alarms[64] := "DB_WinCCAlarms"."1-IO"."1252_HBL_TT_28_Fault".Memory.%X0;
   "DB_Application".FromHB.Alarms[65] := "DB_WinCCAlarms"."1-IO"."1253_HBL_TT_29_Fault".Memory.%X0;
   "DB_Application".FromHB.Alarms[66] := "DB_WinCCAlarms"."1-IO"."1254_HBL_TT_32_Fault".Memory.%X0;
   "DB_Application".FromHB.Alarms[67] := "DB_WinCCAlarms"."1-IO"."1255_HBL_CT_01_Fault".Memory.%X0;
   "DB_Application".FromHB.Alarms[68] := "DB_WinCCAlarms"."1-IO"."1256_HBL_CT_02_Fault".Memory.%X0;
   "DB_Application".FromHB.Alarms[69] := FALSE;
   "DB_Application".FromHB.Alarms[70] := "DB_WinCCAlarms"."1-IO"."1258_HBL_TT_26_Fault".Memory.%X0;
   "DB_Application".FromHB.Alarms[71] := "DB_WinCCAlarms"."1-IO"."1259_HBL_TT_27_Fault".Memory.%X0;
   "DB_Application".FromHB.Alarms[72] := "DB_WinCCAlarms"."1-IO"."1260_HBL_FT_01_Fault".Memory.%X0;
   "DB_Application".FromHB.Alarms[73] := FALSE;
   "DB_Application".FromHB.Alarms[74] := "DB_WinCCAlarms"."1-IO"."1262_HBL_TT_30_Fault".Memory.%X0;
   "DB_Application".FromHB.Alarms[75] := "DB_WinCCAlarms"."1-IO"."1263_HBL_TT_34_Fault".Memory.%X0;
   "DB_Application".FromHB.Alarms[76] := "DB_WinCCAlarms"."1-IO"."1264".Memory.%X0;
END_REGION

REGION Network 7 (SCL): Alarms to App PLC - Group 2
   "DB_Application".FromHB.Alarms[77] := "DB_WinCCAlarms"."2-ProcessValues"."2018".Memory.%X0;
   "DB_Application".FromHB.Alarms[78] := "DB_WinCCAlarms"."2-ProcessValues"."2028".Memory.%X0;
   "DB_Application".FromHB.Alarms[79] := "DB_WinCCAlarms"."2-ProcessValues"."2058".Memory.%X0;
   "DB_Application".FromHB.Alarms[80] := "DB_WinCCAlarms"."2-ProcessValues"."2100".Memory.%X0;
   "DB_Application".FromHB.Alarms[81] := "DB_WinCCAlarms"."2-ProcessValues"."2101".Memory.%X0;
   "DB_Application".FromHB.Alarms[82] := "DB_WinCCAlarms"."2-ProcessValues"."2102".Memory.%X0;
   "DB_Application".FromHB.Alarms[83] := "DB_WinCCAlarms"."2-ProcessValues"."2103".Memory.%X0;
   "DB_Application".FromHB.Alarms[84] := "DB_WinCCAlarms"."2-ProcessValues"."2105".Memory.%X0;
   "DB_Application".FromHB.Alarms[85] := "DB_WinCCAlarms"."2-ProcessValues"."2106".Memory.%X0;
   "DB_Application".FromHB.Alarms[86] := "DB_WinCCAlarms"."2-ProcessValues"."2107".Memory.%X0;
   "DB_Application".FromHB.Alarms[87] := "DB_WinCCAlarms"."2-ProcessValues"."2108".Memory.%X0;
   "DB_Application".FromHB.Alarms[88] := "DB_WinCCAlarms"."2-ProcessValues"."2109".Memory.%X0;
   "DB_Application".FromHB.Alarms[89] := "DB_WinCCAlarms"."2-ProcessValues"."2110".Memory.%X0;
   "DB_Application".FromHB.Alarms[90] := "DB_WinCCAlarms"."2-ProcessValues"."2111".Memory.%X0;
   "DB_Application".FromHB.Alarms[91] := "DB_WinCCAlarms"."2-ProcessValues"."2112".Memory.%X0;
   "DB_Application".FromHB.Alarms[92] := "DB_WinCCAlarms"."2-ProcessValues"."2113".Memory.%X0;
   "DB_Application".FromHB.Alarms[93] := "DB_WinCCAlarms"."2-ProcessValues"."2114".Memory.%X0;
   "DB_Application".FromHB.Alarms[94] := "DB_WinCCAlarms"."2-ProcessValues"."2115".Memory.%X0;
   "DB_Application".FromHB.Alarms[95] := "DB_WinCCAlarms"."2-ProcessValues"."2116".Memory.%X0;
   "DB_Application".FromHB.Alarms[96] := "DB_WinCCAlarms"."2-ProcessValues"."2117".Memory.%X0;
   "DB_Application".FromHB.Alarms[97] := "DB_WinCCAlarms"."2-ProcessValues"."2301_HeatSourceTempDropCritical".Memory.%X0;
   "DB_Application".FromHB.Alarms[98] := "DB_WinCCAlarms"."2-ProcessValues"."2302_HeatSourceTempRiseCritical".Memory.%X0;
   "DB_Application".FromHB.Alarms[99] := "DB_WinCCAlarms"."2-ProcessValues"."2303_SuperheatCompressorHigh".Memory.%X0;
   "DB_Application".FromHB.Alarms[100] := "DB_WinCCAlarms"."2-ProcessValues"."2304_SuperheatCompressorLow".Memory.%X0;
   "DB_Application".FromHB.Alarms[101] := "DB_WinCCAlarms"."2-ProcessValues"."2305_OilFilterDeltaPHigh".Memory.%X0;
   "DB_Application".FromHB.Alarms[102] := "DB_WinCCAlarms"."2-ProcessValues"."2306_OilFilterDeltaPHighHigh".Memory.%X0;
   "DB_Application".FromHB.Alarms[103] := "DB_WinCCAlarms"."2-ProcessValues"."2307_EvaporatorDischargePressureMeanValue".Memory.%X0;
   "DB_Application".FromHB.Alarms[104] := "DB_WinCCAlarms"."2-ProcessValues"."2308_EvaporatorDischargePressureHigh".Memory.%X0;
END_REGION

REGION Network 8 (SCL): Alarms to App PLC - Group 3 & 5
   // Group 3-Control
   "DB_Application".FromHB.Alarms[105] := FALSE; // 3000
   "DB_Application".FromHB.Alarms[106] := "DB_WinCCAlarms"."3-Control"."3020".Memory.%X0;
   "DB_Application".FromHB.Alarms[107] := FALSE; // 3030
   "DB_Application".FromHB.Alarms[108] := FALSE; // 3040
   "DB_Application".FromHB.Alarms[109] := FALSE; // 3050
   "DB_Application".FromHB.Alarms[110] := FALSE; // 3060
   "DB_Application".FromHB.Alarms[111] := FALSE; // 3070
   "DB_Application".FromHB.Alarms[112] := FALSE; // 3080
   "DB_Application".FromHB.Alarms[113] := FALSE; // 3090
   "DB_Application".FromHB.Alarms[114] := FALSE; // 3100
   "DB_Application".FromHB.Alarms[115] := FALSE; // 3110
   "DB_Application".FromHB.Alarms[116] := "DB_WinCCAlarms"."3-Control"."3400_HydrolockProtectionActive".Memory.%X0;
   "DB_Application".FromHB.Alarms[158] := "DB_WinCCAlarms"."3-Control"."3401_DripPanLevelHigh".Memory.%X0;

   // Group 5-Auxiliaries
   "DB_Application".FromHB.Alarms[117] := "DB_WinCCAlarms"."5-Auxiliaries"."5000_OilHeatingActivationFailure".Memory.%X0;
   "DB_Application".FromHB.Alarms[118] := "DB_WinCCAlarms"."5-Auxiliaries"."5001_OilHeatingDeactivationFailure".Memory.%X0;
   "DB_Application".FromHB.Alarms[119] := "DB_WinCCAlarms"."5-Auxiliaries"."5200".Memory.%X0;
   "DB_Application".FromHB.Alarms[120] := "DB_WinCCAlarms"."5-Auxiliaries"."5201".Memory.%X0;
   "DB_Application".FromHB.Alarms[121] := "DB_WinCCAlarms"."5-Auxiliaries"."5202".Memory.%X0;
   "DB_Application".FromHB.Alarms[122] := "DB_WinCCAlarms"."5-Auxiliaries"."5203_CPC_SC_01_CommError".Memory.%X0;
   "DB_Application".FromHB.Alarms[123] := "DB_WinCCAlarms"."5-Auxiliaries"."5204_CPC_SC_01_Tripped".Memory.%X0;
   "DB_Application".FromHB.Alarms[124] := "DB_WinCCAlarms"."5-Auxiliaries"."5205".Memory.%X0;
   "DB_Application".FromHB.Alarms[125] := "DB_WinCCAlarms"."5-Auxiliaries"."5206".Memory.%X0;
   "DB_Application".FromHB.Alarms[126] := "DB_WinCCAlarms"."5-Auxiliaries"."5250_SSC_TT_01_Fault".Memory.%X0;
   "DB_Application".FromHB.Alarms[127] := "DB_WinCCAlarms"."5-Auxiliaries"."5251_SSC_TT_02_Fault".Memory.%X0;
   "DB_Application".FromHB.Alarms[128] := "DB_WinCCAlarms"."5-Auxiliaries"."5252_SSC_TT_03_Fault".Memory.%X0;
   "DB_Application".FromHB.Alarms[129] := "DB_WinCCAlarms"."5-Auxiliaries"."5253_SSC_TT_04_Fault".Memory.%X0;
   "DB_Application".FromHB.Alarms[130] := "DB_WinCCAlarms"."5-Auxiliaries"."5254_SSC_PIT_01_Fault".Memory.%X0;
   "DB_Application".FromHB.Alarms[131] := "DB_WinCCAlarms"."5-Auxiliaries"."5255_SSC_PDT_01_Fault".Memory.%X0;
   "DB_Application".FromHB.Alarms[132] := "DB_WinCCAlarms"."5-Auxiliaries"."5256_SSC_LT_01_Fault".Memory.%X0;
   "DB_Application".FromHB.Alarms[133] := "DB_WinCCAlarms"."5-Auxiliaries"."5257_SSC_LT_01_Low".Memory.%X0;
   "DB_Application".FromHB.Alarms[134] := "DB_WinCCAlarms"."5-Auxiliaries"."5258_SSC_PDT_01_High".Memory.%X0;
   "DB_Application".FromHB.Alarms[135] := "DB_WinCCAlarms"."5-Auxiliaries"."5259_SSC_TT_02_High".Memory.%X0;
   "DB_Application".FromHB.Alarms[136] := "DB_WinCCAlarms"."5-Auxiliaries"."5260_SSC_TT_03_Low".Memory.%X0;
   "DB_Application".FromHB.Alarms[137] := "DB_WinCCAlarms"."5-Auxiliaries"."5261_SSC_PIT_01_Low".Memory.%X0;
   "DB_Application".FromHB.Alarms[138] := "DB_WinCCAlarms"."5-Auxiliaries"."5262_DeltaT_ShaftSealHigh".Memory.%X0;
   "DB_Application".FromHB.Alarms[139] := "DB_WinCCAlarms"."5-Auxiliaries"."5263_SSC_PIT_01_High".Memory.%X0;
   "DB_Application".FromHB.Alarms[140] := "DB_WinCCAlarms"."5-Auxiliaries"."5268_ShaftSealSystemShutdown".Memory.%X0;
END_REGION

REGION Network 9 (SCL): Alarms to App PLC - Group 8
   // Group 8-Events
   //"DB_Application".Status.Alarms[141] := "DB_WinCCAlarms"."8-Events"."8000_State0_Initialize".Memory.%X0;
   //"DB_Application".Status.Alarms[142] := "DB_WinCCAlarms"."8-Events"."8001_State1_Offline".Memory.%X0;
   "DB_Application".FromHB.Alarms[143] := "DB_WinCCAlarms"."8-Events"."8002_State2_Standby".Memory.%X0;
END_REGION
END_FUNCTION_BLOCK

FUNCTION_BLOCK "AlarmManagement"   // FB32, LAD
{ S7_Optimized_Access := 'TRUE' }
VERSION : 0.1
// stored: AutoNumber true, IsIECCheckEnabled false, IsRetainMemResEnabled false, MemoryReserve 0, SetENOAutomatically false, UDAEnableTagReadback false
   VAR
      CriticalAlarm_1000 { ExternalAccessible := 'False'; ExternalVisible := 'False'; ExternalWritable := 'False'} : Bool;   // Contribution from 1000-series
      CriticalAlarm_2000 { ExternalAccessible := 'False'; ExternalVisible := 'False'; ExternalWritable := 'False'} : Bool;   // Contribution from 2000-series
      CriticalAlarm_3000 { ExternalAccessible := 'False'; ExternalVisible := 'False'; ExternalWritable := 'False'} : Bool;   // Contribution from 3000-series
      CriticalAlarm_4000 { ExternalAccessible := 'False'; ExternalVisible := 'False'; ExternalWritable := 'False'} : Bool;   // Contribution from 4000-series
      CriticalAlarm_5000 { ExternalAccessible := 'False'; ExternalVisible := 'False'; ExternalWritable := 'False'} : Bool;   // Contribution from 5000-series
      CriticalAlarm_9000 { ExternalAccessible := 'False'; ExternalVisible := 'False'; ExternalWritable := 'False'} : Bool;   // Contribution from 9000-series
      CommonAlarm_1000 { ExternalAccessible := 'False'; ExternalVisible := 'False'; ExternalWritable := 'False'} : Bool;
      CommonAlarm_2000 { ExternalAccessible := 'False'; ExternalVisible := 'False'; ExternalWritable := 'False'} : Bool;
      CommonAlarm_3000 { ExternalAccessible := 'False'; ExternalVisible := 'False'; ExternalWritable := 'False'} : Bool;
      CommonAlarm_5000 { ExternalAccessible := 'False'; ExternalVisible := 'False'; ExternalWritable := 'False'} : Bool;
      CommonAlarm_9000 { ExternalAccessible := 'False'; ExternalVisible := 'False'; ExternalWritable := 'False'} : Bool;
   END_VAR
BEGIN

REGION Network 1 (SCL): Comments
   (*
   This is done with ladder code instead of bits in an alarm struct, so that:
   a) it is easy to see at a glance which alarms are part of the critical alarm (and when monitoring, which alarms are causing the critical alarm)
   b) alarms cannot be removed from the critical alarm by accidentally flipping a bit in a struct, only via code change

   When adding alarms, please add into the correct group and keep each group ordered by alarm number. You will thank yourself later.
   It is easy to make a mess here, resist the urge!
   *)
END_REGION

REGION Network 2: Critical Alarm 1000
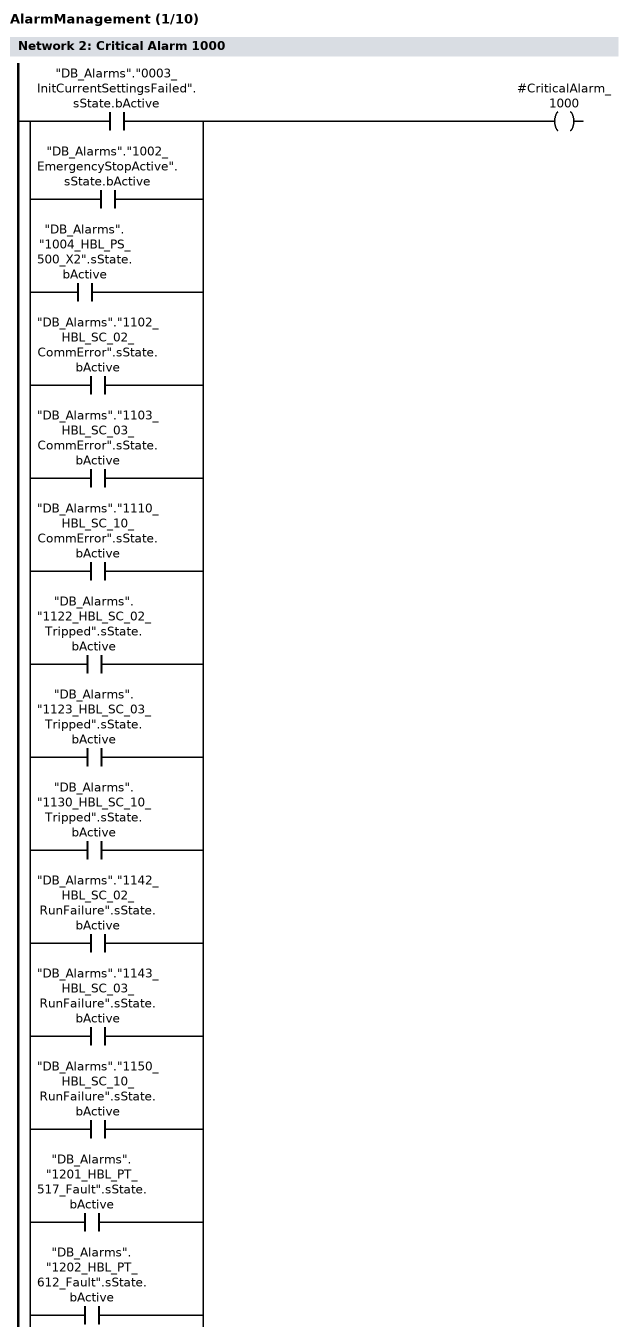
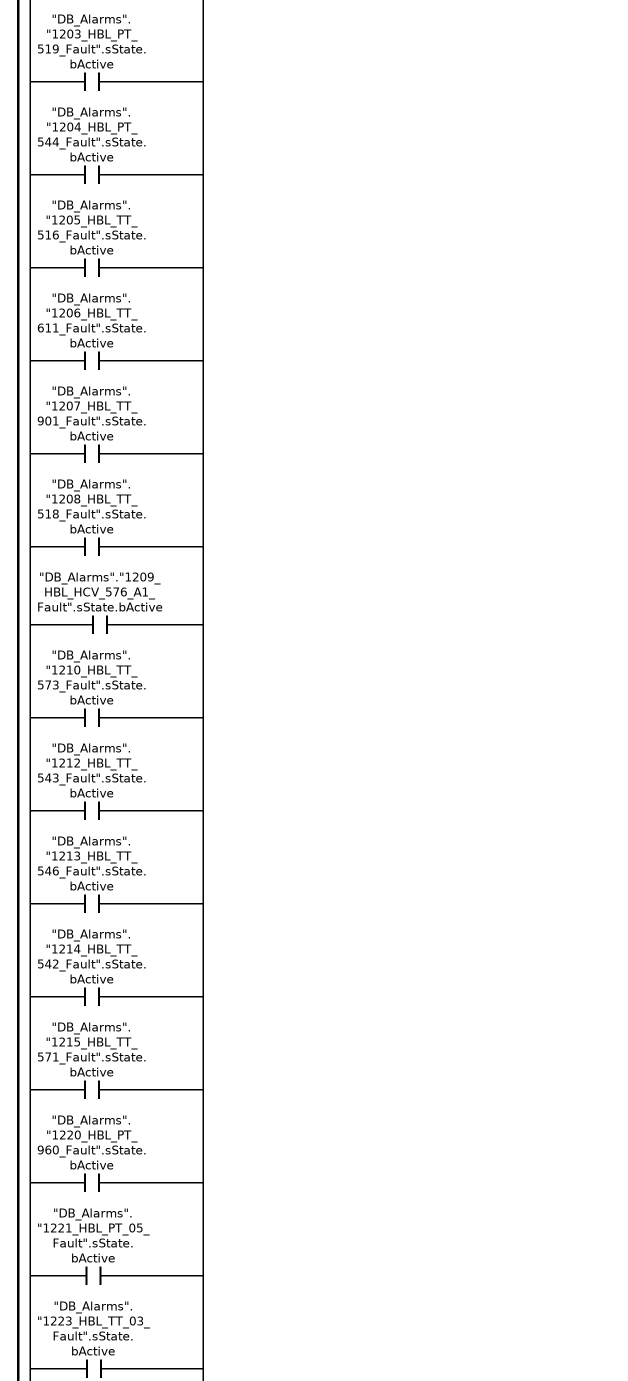
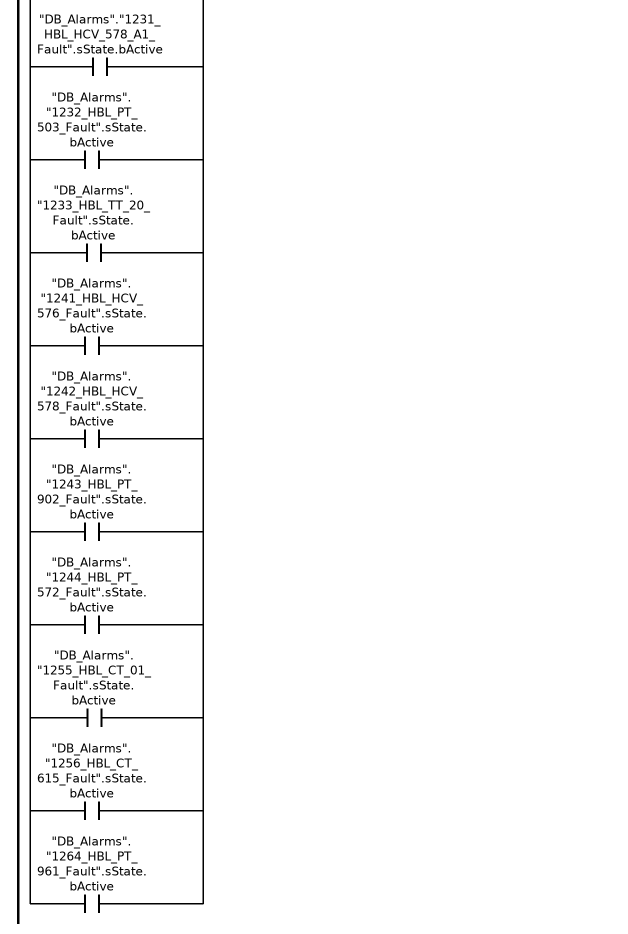
   RUNG wire#powerrail
      Contact( "DB_Alarms"."0003_InitCurrentSettingsFailed".sState.bActive )
      wire#w1
      Coil( #CriticalAlarm_1000 )
   END_RUNG
   RUNG wire#powerrail
      Contact( "DB_Alarms"."1002_EmergencyStopActive".sState.bActive )
   END_RUNG wire#w1
   RUNG wire#powerrail
      Contact( "DB_Alarms"."1004_HBL_PS_500_X2".sState.bActive )
   END_RUNG wire#w1
   RUNG wire#powerrail
      Contact( "DB_Alarms"."1102_HBL_SC_02_CommError".sState.bActive )
   END_RUNG wire#w1
   RUNG wire#powerrail
      Contact( "DB_Alarms"."1103_HBL_SC_03_CommError".sState.bActive )
   END_RUNG wire#w1
   RUNG wire#powerrail
      Contact( "DB_Alarms"."1110_HBL_SC_10_CommError".sState.bActive )
   END_RUNG wire#w1
   RUNG wire#powerrail
      Contact( "DB_Alarms"."1122_HBL_SC_02_Tripped".sState.bActive )
   END_RUNG wire#w1
   RUNG wire#powerrail
      Contact( "DB_Alarms"."1123_HBL_SC_03_Tripped".sState.bActive )
   END_RUNG wire#w1
   RUNG wire#powerrail
      Contact( "DB_Alarms"."1130_HBL_SC_10_Tripped".sState.bActive )
   END_RUNG wire#w1
   RUNG wire#powerrail
      Contact( "DB_Alarms"."1142_HBL_SC_02_RunFailure".sState.bActive )
   END_RUNG wire#w1
   RUNG wire#powerrail
      Contact( "DB_Alarms"."1143_HBL_SC_03_RunFailure".sState.bActive )
   END_RUNG wire#w1
   RUNG wire#powerrail
      Contact( "DB_Alarms"."1150_HBL_SC_10_RunFailure".sState.bActive )
   END_RUNG wire#w1
   RUNG wire#powerrail
      Contact( "DB_Alarms"."1201_HBL_PT_517_Fault".sState.bActive )
   END_RUNG wire#w1
   RUNG wire#powerrail
      Contact( "DB_Alarms"."1202_HBL_PT_612_Fault".sState.bActive )
   END_RUNG wire#w1
   RUNG wire#powerrail
      Contact( "DB_Alarms"."1203_HBL_PT_519_Fault".sState.bActive )
   END_RUNG wire#w1
   RUNG wire#powerrail
      Contact( "DB_Alarms"."1204_HBL_PT_544_Fault".sState.bActive )
   END_RUNG wire#w1
   RUNG wire#powerrail
      Contact( "DB_Alarms"."1205_HBL_TT_516_Fault".sState.bActive )
   END_RUNG wire#w1
   RUNG wire#powerrail
      Contact( "DB_Alarms"."1206_HBL_TT_611_Fault".sState.bActive )
   END_RUNG wire#w1
   RUNG wire#powerrail
      Contact( "DB_Alarms"."1207_HBL_TT_901_Fault".sState.bActive )
   END_RUNG wire#w1
   RUNG wire#powerrail
      Contact( "DB_Alarms"."1208_HBL_TT_518_Fault".sState.bActive )
   END_RUNG wire#w1
   RUNG wire#powerrail
      Contact( "DB_Alarms"."1209_HBL_HCV_576_A1_Fault".sState.bActive )
   END_RUNG wire#w1
   RUNG wire#powerrail
      Contact( "DB_Alarms"."1210_HBL_TT_573_Fault".sState.bActive )
   END_RUNG wire#w1
   RUNG wire#powerrail
      Contact( "DB_Alarms"."1212_HBL_TT_543_Fault".sState.bActive )
   END_RUNG wire#w1
   RUNG wire#powerrail
      Contact( "DB_Alarms"."1213_HBL_TT_546_Fault".sState.bActive )
   END_RUNG wire#w1
   RUNG wire#powerrail
      Contact( "DB_Alarms"."1214_HBL_TT_542_Fault".sState.bActive )
   END_RUNG wire#w1
   RUNG wire#powerrail
      Contact( "DB_Alarms"."1215_HBL_TT_571_Fault".sState.bActive )
   END_RUNG wire#w1
   RUNG wire#powerrail
      Contact( "DB_Alarms"."1220_HBL_PT_960_Fault".sState.bActive )
   END_RUNG wire#w1
   RUNG wire#powerrail
      Contact( "DB_Alarms"."1221_HBL_PT_05_Fault".sState.bActive )
   END_RUNG wire#w1
   RUNG wire#powerrail
      Contact( "DB_Alarms"."1223_HBL_TT_03_Fault".sState.bActive )
   END_RUNG wire#w1
   RUNG wire#powerrail
      Contact( "DB_Alarms"."1231_HBL_HCV_578_A1_Fault".sState.bActive )
   END_RUNG wire#w1
   RUNG wire#powerrail
      Contact( "DB_Alarms"."1232_HBL_PT_503_Fault".sState.bActive )
   END_RUNG wire#w1
   RUNG wire#powerrail
      Contact( "DB_Alarms"."1233_HBL_TT_20_Fault".sState.bActive )
   END_RUNG wire#w1
   RUNG wire#powerrail
      Contact( "DB_Alarms"."1241_HBL_HCV_576_Fault".sState.bActive )
   END_RUNG wire#w1
   RUNG wire#powerrail
      Contact( "DB_Alarms"."1242_HBL_HCV_578_Fault".sState.bActive )
   END_RUNG wire#w1
   RUNG wire#powerrail
      Contact( "DB_Alarms"."1243_HBL_PT_902_Fault".sState.bActive )
   END_RUNG wire#w1
   RUNG wire#powerrail
      Contact( "DB_Alarms"."1244_HBL_PT_572_Fault".sState.bActive )
   END_RUNG wire#w1
   RUNG wire#powerrail
      Contact( "DB_Alarms"."1255_HBL_CT_01_Fault".sState.bActive )
   END_RUNG wire#w1
   RUNG wire#powerrail
      Contact( "DB_Alarms"."1256_HBL_CT_615_Fault".sState.bActive )
   END_RUNG wire#w1
   RUNG wire#powerrail
      Contact( "DB_Alarms"."1264_HBL_PT_961_Fault".sState.bActive )
   END_RUNG wire#w1
   // the same network as SCL:
   #CriticalAlarm_1000 := "DB_Alarms"."0003_InitCurrentSettingsFailed".sState.bActive OR "DB_Alarms"."1002_EmergencyStopActive".sState.bActive OR "DB_Alarms"."1004_HBL_PS_500_X2".sState.bActive OR "DB_Alarms"."1102_HBL_SC_02_CommError".sState.bActive OR "DB_Alarms"."1103_HBL_SC_03_CommError".sState.bActive OR "DB_Alarms"."1110_HBL_SC_10_CommError".sState.bActive OR "DB_Alarms"."1122_HBL_SC_02_Tripped".sState.bActive OR "DB_Alarms"."1123_HBL_SC_03_Tripped".sState.bActive OR "DB_Alarms"."1130_HBL_SC_10_Tripped".sState.bActive OR "DB_Alarms"."1142_HBL_SC_02_RunFailure".sState.bActive OR "DB_Alarms"."1143_HBL_SC_03_RunFailure".sState.bActive OR "DB_Alarms"."1150_HBL_SC_10_RunFailure".sState.bActive OR "DB_Alarms"."1201_HBL_PT_517_Fault".sState.bActive OR "DB_Alarms"."1202_HBL_PT_612_Fault".sState.bActive OR "DB_Alarms"."1203_HBL_PT_519_Fault".sState.bActive OR "DB_Alarms"."1204_HBL_PT_544_Fault".sState.bActive OR "DB_Alarms"."1205_HBL_TT_516_Fault".sState.bActive OR "DB_Alarms"."1206_HBL_TT_611_Fault".sState.bActive OR "DB_Alarms"."1207_HBL_TT_901_Fault".sState.bActive OR "DB_Alarms"."1208_HBL_TT_518_Fault".sState.bActive OR "DB_Alarms"."1209_HBL_HCV_576_A1_Fault".sState.bActive OR "DB_Alarms"."1210_HBL_TT_573_Fault".sState.bActive OR "DB_Alarms"."1212_HBL_TT_543_Fault".sState.bActive OR "DB_Alarms"."1213_HBL_TT_546_Fault".sState.bActive OR "DB_Alarms"."1214_HBL_TT_542_Fault".sState.bActive OR "DB_Alarms"."1215_HBL_TT_571_Fault".sState.bActive OR "DB_Alarms"."1220_HBL_PT_960_Fault".sState.bActive OR "DB_Alarms"."1221_HBL_PT_05_Fault".sState.bActive OR "DB_Alarms"."1223_HBL_TT_03_Fault".sState.bActive OR "DB_Alarms"."1231_HBL_HCV_578_A1_Fault".sState.bActive OR "DB_Alarms"."1232_HBL_PT_503_Fault".sState.bActive OR "DB_Alarms"."1233_HBL_TT_20_Fault".sState.bActive OR "DB_Alarms"."1241_HBL_HCV_576_Fault".sState.bActive OR "DB_Alarms"."1242_HBL_HCV_578_Fault".sState.bActive OR "DB_Alarms"."1243_HBL_PT_902_Fault".sState.bActive OR "DB_Alarms"."1244_HBL_PT_572_Fault".sState.bActive OR "DB_Alarms"."1255_HBL_CT_01_Fault".sState.bActive OR "DB_Alarms"."1256_HBL_CT_615_Fault".sState.bActive OR "DB_Alarms"."1264_HBL_PT_961_Fault".sState.bActive;
END_REGION

REGION Network 3: Critical Alarm 2000
